Fanuc TP program (LS listing): model4_recl.ls

/PROG  model4_recl
/ATTR
COMMENT	= "19-03-19 17:59:41";
PROG_SIZE	= 0;
DEFAULT_GROUP	= 1, *, *, *, *;
/APPL
    ARC Welding Equipment: 1, *, *, *, *;
/MN
   1:  CALL HOME_ALL;
   1:  UFRAME_NUM = 1;
   1:  UTOOL_NUM = 3;
   1:  COL GUARD ADJUST 150;
   1:  PR[91] = PR[90];
   1:  PR[91,1] = PR[90,1] + 6.250;
   1:  PR[91,2] = PR[90,2] + 41.867;
   1:  PR[91,3] = PR[90,3] + 1.495;
   1:  PR[92] = PR[91];
   1:  PR[92,3] = PR[92,3] + 50;
   1:J PR[92] 10% FINE;
   1:L PR[91] R[100]mm/sec CNT100;
   1:  CALL LASER_DRAHT_START;
   1:  PR[91,1] = PR[90,1] + 5.356;
   1:  PR[91,2] = PR[90,2] + 42.761;
   1:L PR[91] R[100]mm/sec CNT100;
   1:  PR[91,1] = PR[90,1] + 3.853;
   1:  PR[91,2] = PR[90,2] + 48.367;
   1:L PR[91] R[100]mm/sec CNT100;
   1:  PR[91,1] = PR[90,1] + 5.356;
   1:  PR[91,2] = PR[90,2] + 53.973;
   1:L PR[91] R[100]mm/sec CNT100;
   1:  PR[91,1] = PR[90,1] + 6.250;
   1:  PR[91,2] = PR[90,2] + 54.867;
   1:L PR[91] R[100]mm/sec CNT100;
   1:  PR[91,1] = PR[90,1] + -1.119;
   1:L PR[91] R[100]mm/sec CNT100;
   1:  PR[91,1] = PR[90,1] + -0.226;
   1:  PR[91,2] = PR[90,2] + 53.973;
   1:L PR[91] R[100]mm/sec CNT100;
   1:  PR[91,1] = PR[90,1] + 1.277;
   1:  PR[91,2] = PR[90,2] + 48.367;
   1:L PR[91] R[100]mm/sec CNT100;
   1:  PR[91,1] = PR[90,1] + -0.226;
   1:  PR[91,2] = PR[90,2] + 42.761;
   1:L PR[91] R[100]mm/sec CNT100;
   1:  PR[91,1] = PR[90,1] + -1.119;
   1:  PR[91,2] = PR[90,2] + 41.867;
   1:L PR[91] R[100]mm/sec CNT100;
   1:  PR[91,1] = PR[90,1] + 6.250;
   1:L PR[91] R[100]mm/sec CNT100TB   .50sec,CALL END_PUD;
   1:  PR[92] = PR[91];
   1:  PR[92,3] = PR[92,3] + 50;
   1:J PR[92] 10% FINE;
   1:  PR[91,1] = PR[90,1] + 25.565;
   1:  PR[91,2] = PR[90,2] + 37.867;
   1:  PR[92] = PR[91];
   1:  PR[92,3] = PR[92,3] + 50;
   1:J PR[92] 10% FINE;
   1:L PR[91] R[100]mm/sec CNT100;
   1:  CALL LASER_DRAHT_START;
   1:  PR[91,2] = PR[90,2] + 58.867;
   1:L PR[91] R[100]mm/sec CNT100;
   1:  PR[91,1] = PR[90,1] + -20.435;
   1:L PR[91] R[100]mm/sec CNT100;
   1:  PR[91,2] = PR[90,2] + 37.867;
   1:L PR[91] R[100]mm/sec CNT100;
   1:  PR[91,1] = PR[90,1] + 25.565;
   1:L PR[91] R[100]mm/sec CNT100TB   .50sec,CALL END_PUD;
   1:  PR[92] = PR[91];
   1:  PR[92,3] = PR[92,3] + 50;
   1:J PR[92] 10% FINE;
   1:  PR[91,1] = PR[90,1] + 18.601;
   1:  PR[91,2] = PR[90,2] + 42.244;
   1:  PR[92] = PR[91];
   1:  PR[92,3] = PR[92,3] + 50;
   1:J PR[92] 10% FINE;
   1:L PR[91] R[100]mm/sec CNT100;
   1:  CALL LASER_DRAHT_START;
   1:  PR[91,1] = PR[90,1] + 15.065;
   1:  PR[91,2] = PR[90,2] + 41.296;
   1:L PR[91] R[100]mm/sec CNT100;
   1:  PR[91,1] = PR[90,1] + 11.530;
   1:  PR[91,2] = PR[90,2] + 42.244;
   1:L PR[91] R[100]mm/sec CNT100;
   1:  PR[91,1] = PR[90,1] + 8.942;
   1:  PR[91,2] = PR[90,2] + 44.831;
   1:L PR[91] R[100]mm/sec CNT100;
   1:  PR[91,1] = PR[90,1] + 7.995;
   1:  PR[91,2] = PR[90,2] + 48.367;
   1:L PR[91] R[100]mm/sec CNT100;
   1:  PR[91,1] = PR[90,1] + 8.942;
   1:  PR[91,2] = PR[90,2] + 51.903;
   1:L PR[91] R[100]mm/sec CNT100;
   1:  PR[91,1] = PR[90,1] + 11.530;
   1:  PR[91,2] = PR[90,2] + 54.490;
   1:L PR[91] R[100]mm/sec CNT100;
   1:  PR[91,1] = PR[90,1] + 15.065;
   1:  PR[91,2] = PR[90,2] + 55.438;
   1:L PR[91] R[100]mm/sec CNT100;
   1:  PR[91,1] = PR[90,1] + 18.601;
   1:  PR[91,2] = PR[90,2] + 54.490;
   1:L PR[91] R[100]mm/sec CNT100;
   1:  PR[91,1] = PR[90,1] + 21.188;
   1:  PR[91,2] = PR[90,2] + 51.903;
   1:L PR[91] R[100]mm/sec CNT100;
   1:  PR[91,1] = PR[90,1] + 22.136;
   1:  PR[91,2] = PR[90,2] + 48.367;
   1:L PR[91] R[100]mm/sec CNT100;
   1:  PR[91,1] = PR[90,1] + 21.188;
   1:  PR[91,2] = PR[90,2] + 44.831;
   1:L PR[91] R[100]mm/sec CNT100;
   1:  PR[91,1] = PR[90,1] + 18.601;
   1:  PR[91,2] = PR[90,2] + 42.244;
   1:L PR[91] R[100]mm/sec CNT100TB   .50sec,CALL END_PUD;
   1:  PR[92] = PR[91];
   1:  PR[92,3] = PR[92,3] + 50;
   1:J PR[92] 10% FINE;
   1:  PR[91,1] = PR[90,1] + -3.812;
   1:  PR[91,2] = PR[90,2] + 44.831;
   1:  PR[92] = PR[91];
   1:  PR[92,3] = PR[92,3] + 50;
   1:J PR[92] 10% FINE;
   1:L PR[91] R[100]mm/sec CNT100;
   1:  CALL LASER_DRAHT_START;
   1:  PR[91,1] = PR[90,1] + -6.399;
   1:  PR[91,2] = PR[90,2] + 42.244;
   1:L PR[91] R[100]mm/sec CNT100;
   1:  PR[91,1] = PR[90,1] + -9.935;
   1:  PR[91,2] = PR[90,2] + 41.296;
   1:L PR[91] R[100]mm/sec CNT100;
   1:  PR[91,1] = PR[90,1] + -13.470;
   1:  PR[91,2] = PR[90,2] + 42.244;
   1:L PR[91] R[100]mm/sec CNT100;
   1:  PR[91,1] = PR[90,1] + -16.058;
   1:  PR[91,2] = PR[90,2] + 44.831;
   1:L PR[91] R[100]mm/sec CNT100;
   1:  PR[91,1] = PR[90,1] + -17.005;
   1:  PR[91,2] = PR[90,2] + 48.367;
   1:L PR[91] R[100]mm/sec CNT100;
   1:  PR[91,1] = PR[90,1] + -16.058;
   1:  PR[91,2] = PR[90,2] + 51.903;
   1:L PR[91] R[100]mm/sec CNT100;
   1:  PR[91,1] = PR[90,1] + -13.470;
   1:  PR[91,2] = PR[90,2] + 54.490;
   1:L PR[91] R[100]mm/sec CNT100;
   1:  PR[91,1] = PR[90,1] + -9.935;
   1:  PR[91,2] = PR[90,2] + 55.438;
   1:L PR[91] R[100]mm/sec CNT100;
   1:  PR[91,1] = PR[90,1] + -6.399;
   1:  PR[91,2] = PR[90,2] + 54.490;
   1:L PR[91] R[100]mm/sec CNT100;
   1:  PR[91,1] = PR[90,1] + -3.812;
   1:  PR[91,2] = PR[90,2] + 51.903;
   1:L PR[91] R[100]mm/sec CNT100;
   1:  PR[91,1] = PR[90,1] + -2.864;
   1:  PR[91,2] = PR[90,2] + 48.367;
   1:L PR[91] R[100]mm/sec CNT100;
   1:  PR[91,1] = PR[90,1] + -3.812;
   1:  PR[91,2] = PR[90,2] + 44.831;
   1:L PR[91] R[100]mm/sec CNT100TB   .50sec,CALL END_PUD;
   1:  PR[92] = PR[91];
   1:  PR[92,3] = PR[92,3] + 50;
   1:J PR[92] 10% FINE;
   1:  PR[91] = PR[90];
   1:  PR[91,1] = PR[90,1] + 6.250;
   1:  PR[91,2] = PR[90,2] + 54.867;
   1:  PR[91,3] = PR[90,3] + 2.795;
   1:  PR[92] = PR[91];
   1:  PR[92,3] = PR[92,3] + 50;
   1:J PR[92] 10% FINE;
   1:L PR[91] R[100]mm/sec CNT100;
   1:  CALL LASER_DRAHT_START;
   1:  PR[91,1] = PR[90,1] + -1.119;
   1:L PR[91] R[100]mm/sec CNT100;
   1:  PR[91,1] = PR[90,1] + -0.226;
   1:  PR[91,2] = PR[90,2] + 53.973;
   1:L PR[91] R[100]mm/sec CNT100;
   1:  PR[91,1] = PR[90,1] + 1.277;
   1:  PR[91,2] = PR[90,2] + 48.367;
   1:L PR[91] R[100]mm/sec CNT100;
   1:  PR[91,1] = PR[90,1] + -0.226;
   1:  PR[91,2] = PR[90,2] + 42.761;
   1:L PR[91] R[100]mm/sec CNT100;
   1:  PR[91,1] = PR[90,1] + -1.119;
   1:  PR[91,2] = PR[90,2] + 41.867;
   1:L PR[91] R[100]mm/sec CNT100;
   1:  PR[91,1] = PR[90,1] + 6.250;
   1:L PR[91] R[100]mm/sec CNT100;
   1:  PR[91,1] = PR[90,1] + 5.356;
   1:  PR[91,2] = PR[90,2] + 42.761;
   1:L PR[91] R[100]mm/sec CNT100;
   1:  PR[91,1] = PR[90,1] + 3.853;
   1:  PR[91,2] = PR[90,2] + 48.367;
   1:L PR[91] R[100]mm/sec CNT100;
   1:  PR[91,1] = PR[90,1] + 5.356;
   1:  PR[91,2] = PR[90,2] + 53.973;
   1:L PR[91] R[100]mm/sec CNT100;
   1:  PR[91,1] = PR[90,1] + 6.250;
   1:  PR[91,2] = PR[90,2] + 54.867;
   1:L PR[91] R[100]mm/sec CNT100TB   .50sec,CALL END_PUD;
   1:  PR[92] = PR[91];
   1:  PR[92,3] = PR[92,3] + 50;
   1:J PR[92] 10% FINE;
   1:  PR[91,1] = PR[90,1] + 25.565;
   1:  PR[91,2] = PR[90,2] + 58.867;
   1:  PR[92] = PR[91];
   1:  PR[92,3] = PR[92,3] + 50;
   1:J PR[92] 10% FINE;
   1:L PR[91] R[100]mm/sec CNT100;
   1:  CALL LASER_DRAHT_START;
   1:  PR[91,1] = PR[90,1] + -20.435;
   1:L PR[91] R[100]mm/sec CNT100;
   1:  PR[91,2] = PR[90,2] + 37.867;
   1:L PR[91] R[100]mm/sec CNT100;
   1:  PR[91,1] = PR[90,1] + 25.565;
   1:L PR[91] R[100]mm/sec CNT100;
   1:  PR[91,2] = PR[90,2] + 58.867;
   1:L PR[91] R[100]mm/sec CNT100TB   .50sec,CALL END_PUD;
   1:  PR[92] = PR[91];
   1:  PR[92,3] = PR[92,3] + 50;
   1:J PR[92] 10% FINE;
   1:  PR[91,1] = PR[90,1] + 18.601;
   1:  PR[91,2] = PR[90,2] + 54.490;
   1:  PR[92] = PR[91];
   1:  PR[92,3] = PR[92,3] + 50;
   1:J PR[92] 10% FINE;
   1:L PR[91] R[100]mm/sec CNT100;
   1:  CALL LASER_DRAHT_START;
   1:  PR[91,1] = PR[90,1] + 21.188;
   1:  PR[91,2] = PR[90,2] + 51.903;
   1:L PR[91] R[100]mm/sec CNT100;
   1:  PR[91,1] = PR[90,1] + 22.136;
   1:  PR[91,2] = PR[90,2] + 48.367;
   1:L PR[91] R[100]mm/sec CNT100;
   1:  PR[91,1] = PR[90,1] + 21.188;
   1:  PR[91,2] = PR[90,2] + 44.831;
   1:L PR[91] R[100]mm/sec CNT100;
   1:  PR[91,1] = PR[90,1] + 18.601;
   1:  PR[91,2] = PR[90,2] + 42.244;
   1:L PR[91] R[100]mm/sec CNT100;
   1:  PR[91,1] = PR[90,1] + 15.065;
   1:  PR[91,2] = PR[90,2] + 41.296;
   1:L PR[91] R[100]mm/sec CNT100;
   1:  PR[91,1] = PR[90,1] + 11.530;
   1:  PR[91,2] = PR[90,2] + 42.244;
   1:L PR[91] R[100]mm/sec CNT100;
   1:  PR[91,1] = PR[90,1] + 8.942;
   1:  PR[91,2] = PR[90,2] + 44.831;
   1:L PR[91] R[100]mm/sec CNT100;
   1:  PR[91,1] = PR[90,1] + 7.995;
   1:  PR[91,2] = PR[90,2] + 48.367;
   1:L PR[91] R[100]mm/sec CNT100;
   1:  PR[91,1] = PR[90,1] + 8.942;
   1:  PR[91,2] = PR[90,2] + 51.903;
   1:L PR[91] R[100]mm/sec CNT100;
   1:  PR[91,1] = PR[90,1] + 11.530;
   1:  PR[91,2] = PR[90,2] + 54.490;
   1:L PR[91] R[100]mm/sec CNT100;
   1:  PR[91,1] = PR[90,1] + 15.065;
   1:  PR[91,2] = PR[90,2] + 55.438;
   1:L PR[91] R[100]mm/sec CNT100;
   1:  PR[91,1] = PR[90,1] + 18.601;
   1:  PR[91,2] = PR[90,2] + 54.490;
   1:L PR[91] R[100]mm/sec CNT100TB   .50sec,CALL END_PUD;
   1:  PR[92] = PR[91];
   1:  PR[92,3] = PR[92,3] + 50;
   1:J PR[92] 10% FINE;
   1:  PR[91,1] = PR[90,1] + -3.812;
   1:  PR[91,2] = PR[90,2] + 51.903;
   1:  PR[92] = PR[91];
   1:  PR[92,3] = PR[92,3] + 50;
   1:J PR[92] 10% FINE;
   1:L PR[91] R[100]mm/sec CNT100;
   1:  CALL LASER_DRAHT_START;
   1:  PR[91,1] = PR[90,1] + -2.864;
   1:  PR[91,2] = PR[90,2] + 48.367;
   1:L PR[91] R[100]mm/sec CNT100;
   1:  PR[91,1] = PR[90,1] + -3.812;
   1:  PR[91,2] = PR[90,2] + 44.831;
   1:L PR[91] R[100]mm/sec CNT100;
   1:  PR[91,1] = PR[90,1] + -6.399;
   1:  PR[91,2] = PR[90,2] + 42.244;
   1:L PR[91] R[100]mm/sec CNT100;
   1:  PR[91,1] = PR[90,1] + -9.935;
   1:  PR[91,2] = PR[90,2] + 41.296;
   1:L PR[91] R[100]mm/sec CNT100;
   1:  PR[91,1] = PR[90,1] + -13.470;
   1:  PR[91,2] = PR[90,2] + 42.244;
   1:L PR[91] R[100]mm/sec CNT100;
   1:  PR[91,1] = PR[90,1] + -16.058;
   1:  PR[91,2] = PR[90,2] + 44.831;
   1:L PR[91] R[100]mm/sec CNT100;
   1:  PR[91,1] = PR[90,1] + -17.005;
   1:  PR[91,2] = PR[90,2] + 48.367;
   1:L PR[91] R[100]mm/sec CNT100;
   1:  PR[91,1] = PR[90,1] + -16.058;
   1:  PR[91,2] = PR[90,2] + 51.903;
   1:L PR[91] R[100]mm/sec CNT100;
   1:  PR[91,1] = PR[90,1] + -13.470;
   1:  PR[91,2] = PR[90,2] + 54.490;
   1:L PR[91] R[100]mm/sec CNT100;
   1:  PR[91,1] = PR[90,1] + -9.935;
   1:  PR[91,2] = PR[90,2] + 55.438;
   1:L PR[91] R[100]mm/sec CNT100;
   1:  PR[91,1] = PR[90,1] + -6.399;
   1:  PR[91,2] = PR[90,2] + 54.490;
   1:L PR[91] R[100]mm/sec CNT100;
   1:  PR[91,1] = PR[90,1] + -3.812;
   1:  PR[91,2] = PR[90,2] + 51.903;
   1:L PR[91] R[100]mm/sec CNT100TB   .50sec,CALL END_PUD;
   1:  PR[92] = PR[91];
   1:  PR[92,3] = PR[92,3] + 50;
   1:J PR[92] 10% FINE;
   1:  PR[91] = PR[90];
   1:  PR[91,1] = PR[90,1] + 6.250;
   1:  PR[91,2] = PR[90,2] + 54.867;
   1:  PR[91,3] = PR[90,3] + 4.095;
   1:  PR[92] = PR[91];
   1:  PR[92,3] = PR[92,3] + 50;
   1:J PR[92] 10% FINE;
   1:L PR[91] R[100]mm/sec CNT100;
   1:  CALL LASER_DRAHT_START;
   1:  PR[91,1] = PR[90,1] + -1.119;
   1:L PR[91] R[100]mm/sec CNT100;
   1:  PR[91,1] = PR[90,1] + -0.226;
   1:  PR[91,2] = PR[90,2] + 53.973;
   1:L PR[91] R[100]mm/sec CNT100;
   1:  PR[91,1] = PR[90,1] + 1.277;
   1:  PR[91,2] = PR[90,2] + 48.367;
   1:L PR[91] R[100]mm/sec CNT100;
   1:  PR[91,1] = PR[90,1] + -0.226;
   1:  PR[91,2] = PR[90,2] + 42.761;
   1:L PR[91] R[100]mm/sec CNT100;
   1:  PR[91,1] = PR[90,1] + -1.119;
   1:  PR[91,2] = PR[90,2] + 41.867;
   1:L PR[91] R[100]mm/sec CNT100;
   1:  PR[91,1] = PR[90,1] + 6.250;
   1:L PR[91] R[100]mm/sec CNT100;
   1:  PR[91,1] = PR[90,1] + 5.356;
   1:  PR[91,2] = PR[90,2] + 42.761;
   1:L PR[91] R[100]mm/sec CNT100;
   1:  PR[91,1] = PR[90,1] + 3.853;
   1:  PR[91,2] = PR[90,2] + 48.367;
   1:L PR[91] R[100]mm/sec CNT100;
   1:  PR[91,1] = PR[90,1] + 5.356;
   1:  PR[91,2] = PR[90,2] + 53.973;
   1:L PR[91] R[100]mm/sec CNT100;
   1:  PR[91,1] = PR[90,1] + 6.250;
   1:  PR[91,2] = PR[90,2] + 54.867;
   1:L PR[91] R[100]mm/sec CNT100TB   .50sec,CALL END_PUD;
   1:  PR[92] = PR[91];
   1:  PR[92,3] = PR[92,3] + 50;
   1:J PR[92] 10% FINE;
   1:  PR[91,1] = PR[90,1] + 25.565;
   1:  PR[91,2] = PR[90,2] + 58.867;
   1:  PR[92] = PR[91];
   1:  PR[92,3] = PR[92,3] + 50;
   1:J PR[92] 10% FINE;
   1:L PR[91] R[100]mm/sec CNT100;
   1:  CALL LASER_DRAHT_START;
   1:  PR[91,1] = PR[90,1] + -20.435;
   1:L PR[91] R[100]mm/sec CNT100;
   1:  PR[91,2] = PR[90,2] + 37.867;
   1:L PR[91] R[100]mm/sec CNT100;
   1:  PR[91,1] = PR[90,1] + 25.565;
   1:L PR[91] R[100]mm/sec CNT100;
   1:  PR[91,2] = PR[90,2] + 58.867;
   1:L PR[91] R[100]mm/sec CNT100TB   .50sec,CALL END_PUD;
   1:  PR[92] = PR[91];
   1:  PR[92,3] = PR[92,3] + 50;
   1:J PR[92] 10% FINE;
   1:  PR[91,1] = PR[90,1] + 21.188;
   1:  PR[91,2] = PR[90,2] + 51.903;
   1:  PR[92] = PR[91];
   1:  PR[92,3] = PR[92,3] + 50;
   1:J PR[92] 10% FINE;
   1:L PR[91] R[100]mm/sec CNT100;
   1:  CALL LASER_DRAHT_START;
   1:  PR[91,1] = PR[90,1] + 22.136;
   1:  PR[91,2] = PR[90,2] + 48.367;
   1:L PR[91] R[100]mm/sec CNT100;
   1:  PR[91,1] = PR[90,1] + 21.188;
   1:  PR[91,2] = PR[90,2] + 44.831;
   1:L PR[91] R[100]mm/sec CNT100;
   1:  PR[91,1] = PR[90,1] + 18.601;
   1:  PR[91,2] = PR[90,2] + 42.244;
   1:L PR[91] R[100]mm/sec CNT100;
   1:  PR[91,1] = PR[90,1] + 15.065;
   1:  PR[91,2] = PR[90,2] + 41.296;
   1:L PR[91] R[100]mm/sec CNT100;
   1:  PR[91,1] = PR[90,1] + 11.530;
   1:  PR[91,2] = PR[90,2] + 42.244;
   1:L PR[91] R[100]mm/sec CNT100;
   1:  PR[91,1] = PR[90,1] + 8.942;
   1:  PR[91,2] = PR[90,2] + 44.831;
   1:L PR[91] R[100]mm/sec CNT100;
   1:  PR[91,1] = PR[90,1] + 7.995;
   1:  PR[91,2] = PR[90,2] + 48.367;
   1:L PR[91] R[100]mm/sec CNT100;
   1:  PR[91,1] = PR[90,1] + 8.942;
   1:  PR[91,2] = PR[90,2] + 51.903;
   1:L PR[91] R[100]mm/sec CNT100;
   1:  PR[91,1] = PR[90,1] + 11.530;
   1:  PR[91,2] = PR[90,2] + 54.490;
   1:L PR[91] R[100]mm/sec CNT100;
   1:  PR[91,1] = PR[90,1] + 15.065;
   1:  PR[91,2] = PR[90,2] + 55.438;
   1:L PR[91] R[100]mm/sec CNT100;
   1:  PR[91,1] = PR[90,1] + 18.601;
   1:  PR[91,2] = PR[90,2] + 54.490;
   1:L PR[91] R[100]mm/sec CNT100;
   1:  PR[91,1] = PR[90,1] + 21.188;
   1:  PR[91,2] = PR[90,2] + 51.903;
   1:L PR[91] R[100]mm/sec CNT100TB   .50sec,CALL END_PUD;
   1:  PR[92] = PR[91];
   1:  PR[92,3] = PR[92,3] + 50;
   1:J PR[92] 10% FINE;
   1:  PR[91,1] = PR[90,1] + -3.812;
   1:  PR[92] = PR[91];
   1:  PR[92,3] = PR[92,3] + 50;
   1:J PR[92] 10% FINE;
   1:L PR[91] R[100]mm/sec CNT100;
   1:  CALL LASER_DRAHT_START;
   1:  PR[91,1] = PR[90,1] + -2.864;
   1:  PR[91,2] = PR[90,2] + 48.367;
   1:L PR[91] R[100]mm/sec CNT100;
   1:  PR[91,1] = PR[90,1] + -3.812;
   1:  PR[91,2] = PR[90,2] + 44.831;
   1:L PR[91] R[100]mm/sec CNT100;
   1:  PR[91,1] = PR[90,1] + -6.399;
   1:  PR[91,2] = PR[90,2] + 42.244;
   1:L PR[91] R[100]mm/sec CNT100;
   1:  PR[91,1] = PR[90,1] + -9.935;
   1:  PR[91,2] = PR[90,2] + 41.296;
   1:L PR[91] R[100]mm/sec CNT100;
   1:  PR[91,1] = PR[90,1] + -13.470;
   1:  PR[91,2] = PR[90,2] + 42.244;
   1:L PR[91] R[100]mm/sec CNT100;
   1:  PR[91,1] = PR[90,1] + -16.058;
   1:  PR[91,2] = PR[90,2] + 44.831;
   1:L PR[91] R[100]mm/sec CNT100;
   1:  PR[91,1] = PR[90,1] + -17.005;
   1:  PR[91,2] = PR[90,2] + 48.367;
   1:L PR[91] R[100]mm/sec CNT100;
   1:  PR[91,1] = PR[90,1] + -16.058;
   1:  PR[91,2] = PR[90,2] + 51.903;
   1:L PR[91] R[100]mm/sec CNT100;
   1:  PR[91,1] = PR[90,1] + -13.470;
   1:  PR[91,2] = PR[90,2] + 54.490;
   1:L PR[91] R[100]mm/sec CNT100;
   1:  PR[91,1] = PR[90,1] + -9.935;
   1:  PR[91,2] = PR[90,2] + 55.438;
   1:L PR[91] R[100]mm/sec CNT100;
   1:  PR[91,1] = PR[90,1] + -6.399;
   1:  PR[91,2] = PR[90,2] + 54.490;
   1:L PR[91] R[100]mm/sec CNT100;
   1:  PR[91,1] = PR[90,1] + -3.812;
   1:  PR[91,2] = PR[90,2] + 51.903;
   1:L PR[91] R[100]mm/sec CNT100TB   .50sec,CALL END_PUD;
   1:  PR[92] = PR[91];
   1:  PR[92,3] = PR[92,3] + 50;
   1:J PR[92] 10% FINE;
   1:  PR[91] = PR[90];
   1:  PR[91,1] = PR[90,1] + -1.119;
   1:  PR[91,2] = PR[90,2] + 41.867;
   1:  PR[91,3] = PR[90,3] + 5.395;
   1:  PR[92] = PR[91];
   1:  PR[92,3] = PR[92,3] + 50;
   1:J PR[92] 10% FINE;
   1:L PR[91] R[100]mm/sec CNT100;
   1:  CALL LASER_DRAHT_START;
   1:  PR[91,1] = PR[90,1] + 6.250;
   1:L PR[91] R[100]mm/sec CNT100;
   1:  PR[91,1] = PR[90,1] + 5.356;
   1:  PR[91,2] = PR[90,2] + 42.761;
   1:L PR[91] R[100]mm/sec CNT100;
   1:  PR[91,1] = PR[90,1] + 3.853;
   1:  PR[91,2] = PR[90,2] + 48.367;
   1:L PR[91] R[100]mm/sec CNT100;
   1:  PR[91,1] = PR[90,1] + 5.356;
   1:  PR[91,2] = PR[90,2] + 53.973;
   1:L PR[91] R[100]mm/sec CNT100;
   1:  PR[91,1] = PR[90,1] + 6.250;
   1:  PR[91,2] = PR[90,2] + 54.867;
   1:L PR[91] R[100]mm/sec CNT100;
   1:  PR[91,1] = PR[90,1] + -1.119;
   1:L PR[91] R[100]mm/sec CNT100;
   1:  PR[91,1] = PR[90,1] + -0.226;
   1:  PR[91,2] = PR[90,2] + 53.973;
   1:L PR[91] R[100]mm/sec CNT100;
   1:  PR[91,1] = PR[90,1] + 1.277;
   1:  PR[91,2] = PR[90,2] + 48.367;
   1:L PR[91] R[100]mm/sec CNT100;
   1:  PR[91,1] = PR[90,1] + -0.226;
   1:  PR[91,2] = PR[90,2] + 42.761;
   1:L PR[91] R[100]mm/sec CNT100;
   1:  PR[91,1] = PR[90,1] + -1.119;
   1:  PR[91,2] = PR[90,2] + 41.867;
   1:L PR[91] R[100]mm/sec CNT100TB   .50sec,CALL END_PUD;
   1:  PR[92] = PR[91];
   1:  PR[92,3] = PR[92,3] + 50;
   1:J PR[92] 10% FINE;
   1:  PR[91,1] = PR[90,1] + -20.435;
   1:  PR[91,2] = PR[90,2] + 37.867;
   1:  PR[92] = PR[91];
   1:  PR[92,3] = PR[92,3] + 50;
   1:J PR[92] 10% FINE;
   1:L PR[91] R[100]mm/sec CNT100;
   1:  CALL LASER_DRAHT_START;
   1:  PR[91,1] = PR[90,1] + 25.565;
   1:L PR[91] R[100]mm/sec CNT100;
   1:  PR[91,2] = PR[90,2] + 58.867;
   1:L PR[91] R[100]mm/sec CNT100;
   1:  PR[91,1] = PR[90,1] + -20.435;
   1:L PR[91] R[100]mm/sec CNT100;
   1:  PR[91,2] = PR[90,2] + 37.867;
   1:L PR[91] R[100]mm/sec CNT100TB   .50sec,CALL END_PUD;
   1:  PR[92] = PR[91];
   1:  PR[92,3] = PR[92,3] + 50;
   1:J PR[92] 10% FINE;
   1:  PR[91,1] = PR[90,1] + -16.058;
   1:  PR[91,2] = PR[90,2] + 44.831;
   1:  PR[92] = PR[91];
   1:  PR[92,3] = PR[92,3] + 50;
   1:J PR[92] 10% FINE;
   1:L PR[91] R[100]mm/sec CNT100;
   1:  CALL LASER_DRAHT_START;
   1:  PR[91,1] = PR[90,1] + -17.005;
   1:  PR[91,2] = PR[90,2] + 48.367;
   1:L PR[91] R[100]mm/sec CNT100;
   1:  PR[91,1] = PR[90,1] + -16.058;
   1:  PR[91,2] = PR[90,2] + 51.903;
   1:L PR[91] R[100]mm/sec CNT100;
   1:  PR[91,1] = PR[90,1] + -13.470;
   1:  PR[91,2] = PR[90,2] + 54.490;
   1:L PR[91] R[100]mm/sec CNT100;
   1:  PR[91,1] = PR[90,1] + -9.935;
   1:  PR[91,2] = PR[90,2] + 55.438;
   1:L PR[91] R[100]mm/sec CNT100;
   1:  PR[91,1] = PR[90,1] + -6.399;
   1:  PR[91,2] = PR[90,2] + 54.490;
   1:L PR[91] R[100]mm/sec CNT100;
   1:  PR[91,1] = PR[90,1] + -3.812;
   1:  PR[91,2] = PR[90,2] + 51.903;
   1:L PR[91] R[100]mm/sec CNT100;
   1:  PR[91,1] = PR[90,1] + -2.864;
   1:  PR[91,2] = PR[90,2] + 48.367;
   1:L PR[91] R[100]mm/sec CNT100;
   1:  PR[91,1] = PR[90,1] + -3.812;
   1:  PR[91,2] = PR[90,2] + 44.831;
   1:L PR[91] R[100]mm/sec CNT100;
   1:  PR[91,1] = PR[90,1] + -6.399;
   1:  PR[91,2] = PR[90,2] + 42.244;
   1:L PR[91] R[100]mm/sec CNT100;
   1:  PR[91,1] = PR[90,1] + -9.935;
   1:  PR[91,2] = PR[90,2] + 41.296;
   1:L PR[91] R[100]mm/sec CNT100;
   1:  PR[91,1] = PR[90,1] + -13.470;
   1:  PR[91,2] = PR[90,2] + 42.244;
   1:L PR[91] R[100]mm/sec CNT100;
   1:  PR[91,1] = PR[90,1] + -16.058;
   1:  PR[91,2] = PR[90,2] + 44.831;
   1:L PR[91] R[100]mm/sec CNT100TB   .50sec,CALL END_PUD;
   1:  PR[92] = PR[91];
   1:  PR[92,3] = PR[92,3] + 50;
   1:J PR[92] 10% FINE;
   1:  PR[91,1] = PR[90,1] + 8.942;
   1:  PR[92] = PR[91];
   1:  PR[92,3] = PR[92,3] + 50;
   1:J PR[92] 10% FINE;
   1:L PR[91] R[100]mm/sec CNT100;
   1:  CALL LASER_DRAHT_START;
   1:  PR[91,1] = PR[90,1] + 7.995;
   1:  PR[91,2] = PR[90,2] + 48.367;
   1:L PR[91] R[100]mm/sec CNT100;
   1:  PR[91,1] = PR[90,1] + 8.942;
   1:  PR[91,2] = PR[90,2] + 51.903;
   1:L PR[91] R[100]mm/sec CNT100;
   1:  PR[91,1] = PR[90,1] + 11.530;
   1:  PR[91,2] = PR[90,2] + 54.490;
   1:L PR[91] R[100]mm/sec CNT100;
   1:  PR[91,1] = PR[90,1] + 15.065;
   1:  PR[91,2] = PR[90,2] + 55.438;
   1:L PR[91] R[100]mm/sec CNT100;
   1:  PR[91,1] = PR[90,1] + 18.601;
   1:  PR[91,2] = PR[90,2] + 54.490;
   1:L PR[91] R[100]mm/sec CNT100;
   1:  PR[91,1] = PR[90,1] + 21.188;
   1:  PR[91,2] = PR[90,2] + 51.903;
   1:L PR[91] R[100]mm/sec CNT100;
   1:  PR[91,1] = PR[90,1] + 22.136;
   1:  PR[91,2] = PR[90,2] + 48.367;
   1:L PR[91] R[100]mm/sec CNT100;
   1:  PR[91,1] = PR[90,1] + 21.188;
   1:  PR[91,2] = PR[90,2] + 44.831;
   1:L PR[91] R[100]mm/sec CNT100;
   1:  PR[91,1] = PR[90,1] + 18.601;
   1:  PR[91,2] = PR[90,2] + 42.244;
   1:L PR[91] R[100]mm/sec CNT100;
   1:  PR[91,1] = PR[90,1] + 15.065;
   1:  PR[91,2] = PR[90,2] + 41.296;
   1:L PR[91] R[100]mm/sec CNT100;
   1:  PR[91,1] = PR[90,1] + 11.530;
   1:  PR[91,2] = PR[90,2] + 42.244;
   1:L PR[91] R[100]mm/sec CNT100;
   1:  PR[91,1] = PR[90,1] + 8.942;
   1:  PR[91,2] = PR[90,2] + 44.831;
   1:L PR[91] R[100]mm/sec CNT100TB   .50sec,CALL END_PUD;
   1:  PR[92] = PR[91];
   1:  PR[92,3] = PR[92,3] + 50;
   1:J PR[92] 10% FINE;
   1:  PR[91] = PR[90];
   1:  PR[91,1] = PR[90,1] + 6.250;
   1:  PR[91,2] = PR[90,2] + 54.867;
   1:  PR[91,3] = PR[90,3] + 6.695;
   1:  PR[92] = PR[91];
   1:  PR[92,3] = PR[92,3] + 50;
   1:J PR[92] 10% FINE;
   1:L PR[91] R[100]mm/sec CNT100;
   1:  CALL LASER_DRAHT_START;
   1:  PR[91,1] = PR[90,1] + -1.119;
   1:L PR[91] R[100]mm/sec CNT100;
   1:  PR[91,1] = PR[90,1] + -0.226;
   1:  PR[91,2] = PR[90,2] + 53.973;
   1:L PR[91] R[100]mm/sec CNT100;
   1:  PR[91,1] = PR[90,1] + 1.277;
   1:  PR[91,2] = PR[90,2] + 48.367;
   1:L PR[91] R[100]mm/sec CNT100;
   1:  PR[91,1] = PR[90,1] + -0.226;
   1:  PR[91,2] = PR[90,2] + 42.761;
   1:L PR[91] R[100]mm/sec CNT100;
   1:  PR[91,1] = PR[90,1] + -1.119;
   1:  PR[91,2] = PR[90,2] + 41.867;
   1:L PR[91] R[100]mm/sec CNT100;
   1:  PR[91,1] = PR[90,1] + 6.250;
   1:L PR[91] R[100]mm/sec CNT100;
   1:  PR[91,1] = PR[90,1] + 5.356;
   1:  PR[91,2] = PR[90,2] + 42.761;
   1:L PR[91] R[100]mm/sec CNT100;
   1:  PR[91,1] = PR[90,1] + 3.853;
   1:  PR[91,2] = PR[90,2] + 48.367;
   1:L PR[91] R[100]mm/sec CNT100;
   1:  PR[91,1] = PR[90,1] + 5.356;
   1:  PR[91,2] = PR[90,2] + 53.973;
   1:L PR[91] R[100]mm/sec CNT100;
   1:  PR[91,1] = PR[90,1] + 6.250;
   1:  PR[91,2] = PR[90,2] + 54.867;
   1:L PR[91] R[100]mm/sec CNT100TB   .50sec,CALL END_PUD;
   1:  PR[92] = PR[91];
   1:  PR[92,3] = PR[92,3] + 50;
   1:J PR[92] 10% FINE;
   1:  PR[91,1] = PR[90,1] + 25.565;
   1:  PR[91,2] = PR[90,2] + 58.867;
   1:  PR[92] = PR[91];
   1:  PR[92,3] = PR[92,3] + 50;
   1:J PR[92] 10% FINE;
   1:L PR[91] R[100]mm/sec CNT100;
   1:  CALL LASER_DRAHT_START;
   1:  PR[91,1] = PR[90,1] + -20.435;
   1:L PR[91] R[100]mm/sec CNT100;
   1:  PR[91,2] = PR[90,2] + 37.867;
   1:L PR[91] R[100]mm/sec CNT100;
   1:  PR[91,1] = PR[90,1] + 25.565;
   1:L PR[91] R[100]mm/sec CNT100;
   1:  PR[91,2] = PR[90,2] + 58.867;
   1:L PR[91] R[100]mm/sec CNT100TB   .50sec,CALL END_PUD;
   1:  PR[92] = PR[91];
   1:  PR[92,3] = PR[92,3] + 50;
   1:J PR[92] 10% FINE;
   1:  PR[91,1] = PR[90,1] + 21.188;
   1:  PR[91,2] = PR[90,2] + 51.903;
   1:  PR[92] = PR[91];
   1:  PR[92,3] = PR[92,3] + 50;
   1:J PR[92] 10% FINE;
   1:L PR[91] R[100]mm/sec CNT100;
   1:  CALL LASER_DRAHT_START;
   1:  PR[91,1] = PR[90,1] + 22.136;
   1:  PR[91,2] = PR[90,2] + 48.367;
   1:L PR[91] R[100]mm/sec CNT100;
   1:  PR[91,1] = PR[90,1] + 21.188;
   1:  PR[91,2] = PR[90,2] + 44.831;
   1:L PR[91] R[100]mm/sec CNT100;
   1:  PR[91,1] = PR[90,1] + 18.601;
   1:  PR[91,2] = PR[90,2] + 42.244;
   1:L PR[91] R[100]mm/sec CNT100;
   1:  PR[91,1] = PR[90,1] + 15.065;
   1:  PR[91,2] = PR[90,2] + 41.296;
   1:L PR[91] R[100]mm/sec CNT100;
   1:  PR[91,1] = PR[90,1] + 11.530;
   1:  PR[91,2] = PR[90,2] + 42.244;
   1:L PR[91] R[100]mm/sec CNT100;
   1:  PR[91,1] = PR[90,1] + 8.942;
   1:  PR[91,2] = PR[90,2] + 44.831;
   1:L PR[91] R[100]mm/sec CNT100;
   1:  PR[91,1] = PR[90,1] + 7.995;
   1:  PR[91,2] = PR[90,2] + 48.367;
   1:L PR[91] R[100]mm/sec CNT100;
   1:  PR[91,1] = PR[90,1] + 8.942;
   1:  PR[91,2] = PR[90,2] + 51.903;
   1:L PR[91] R[100]mm/sec CNT100;
   1:  PR[91,1] = PR[90,1] + 11.530;
   1:  PR[91,2] = PR[90,2] + 54.490;
   1:L PR[91] R[100]mm/sec CNT100;
   1:  PR[91,1] = PR[90,1] + 15.065;
   1:  PR[91,2] = PR[90,2] + 55.438;
   1:L PR[91] R[100]mm/sec CNT100;
   1:  PR[91,1] = PR[90,1] + 18.601;
   1:  PR[91,2] = PR[90,2] + 54.490;
   1:L PR[91] R[100]mm/sec CNT100;
   1:  PR[91,1] = PR[90,1] + 21.188;
   1:  PR[91,2] = PR[90,2] + 51.903;
   1:L PR[91] R[100]mm/sec CNT100TB   .50sec,CALL END_PUD;
   1:  PR[92] = PR[91];
   1:  PR[92,3] = PR[92,3] + 50;
   1:J PR[92] 10% FINE;
   1:  PR[91,1] = PR[90,1] + -3.812;
   1:  PR[92] = PR[91];
   1:  PR[92,3] = PR[92,3] + 50;
   1:J PR[92] 10% FINE;
   1:L PR[91] R[100]mm/sec CNT100;
   1:  CALL LASER_DRAHT_START;
   1:  PR[91,1] = PR[90,1] + -2.864;
   1:  PR[91,2] = PR[90,2] + 48.367;
   1:L PR[91] R[100]mm/sec CNT100;
   1:  PR[91,1] = PR[90,1] + -3.812;
   1:  PR[91,2] = PR[90,2] + 44.831;
   1:L PR[91] R[100]mm/sec CNT100;
   1:  PR[91,1] = PR[90,1] + -6.399;
   1:  PR[91,2] = PR[90,2] + 42.244;
   1:L PR[91] R[100]mm/sec CNT100;
   1:  PR[91,1] = PR[90,1] + -9.935;
   1:  PR[91,2] = PR[90,2] + 41.296;
   1:L PR[91] R[100]mm/sec CNT100;
   1:  PR[91,1] = PR[90,1] + -13.470;
   1:  PR[91,2] = PR[90,2] + 42.244;
   1:L PR[91] R[100]mm/sec CNT100;
   1:  PR[91,1] = PR[90,1] + -16.058;
   1:  PR[91,2] = PR[90,2] + 44.831;
   1:L PR[91] R[100]mm/sec CNT100;
   1:  PR[91,1] = PR[90,1] + -17.005;
   1:  PR[91,2] = PR[90,2] + 48.367;
   1:L PR[91] R[100]mm/sec CNT100;
   1:  PR[91,1] = PR[90,1] + -16.058;
   1:  PR[91,2] = PR[90,2] + 51.903;
   1:L PR[91] R[100]mm/sec CNT100;
   1:  PR[91,1] = PR[90,1] + -13.470;
   1:  PR[91,2] = PR[90,2] + 54.490;
   1:L PR[91] R[100]mm/sec CNT100;
   1:  PR[91,1] = PR[90,1] + -9.935;
   1:  PR[91,2] = PR[90,2] + 55.438;
   1:L PR[91] R[100]mm/sec CNT100;
   1:  PR[91,1] = PR[90,1] + -6.399;
   1:  PR[91,2] = PR[90,2] + 54.490;
   1:L PR[91] R[100]mm/sec CNT100;
   1:  PR[91,1] = PR[90,1] + -3.812;
   1:  PR[91,2] = PR[90,2] + 51.903;
   1:L PR[91] R[100]mm/sec CNT100TB   .50sec,CALL END_PUD;
   1:  PR[92] = PR[91];
   1:  PR[92,3] = PR[92,3] + 50;
   1:J PR[92] 10% FINE;
   1:  PR[91] = PR[90];
   1:  PR[91,1] = PR[90,1] + -1.119;
   1:  PR[91,2] = PR[90,2] + 54.867;
   1:  PR[91,3] = PR[90,3] + 7.995;
   1:  PR[92] = PR[91];
   1:  PR[92,3] = PR[92,3] + 50;
   1:J PR[92] 10% FINE;
   1:L PR[91] R[100]mm/sec CNT100;
   1:  CALL LASER_DRAHT_START;
   1:  PR[91,1] = PR[90,1] + -0.226;
   1:  PR[91,2] = PR[90,2] + 53.973;
   1:L PR[91] R[100]mm/sec CNT100;
   1:  PR[91,1] = PR[90,1] + 1.277;
   1:  PR[91,2] = PR[90,2] + 48.367;
   1:L PR[91] R[100]mm/sec CNT100;
   1:  PR[91,1] = PR[90,1] + -0.226;
   1:  PR[91,2] = PR[90,2] + 42.761;
   1:L PR[91] R[100]mm/sec CNT100;
   1:  PR[91,1] = PR[90,1] + -1.119;
   1:  PR[91,2] = PR[90,2] + 41.867;
   1:L PR[91] R[100]mm/sec CNT100;
   1:  PR[91,1] = PR[90,1] + 6.250;
   1:L PR[91] R[100]mm/sec CNT100;
   1:  PR[91,1] = PR[90,1] + 5.356;
   1:  PR[91,2] = PR[90,2] + 42.761;
   1:L PR[91] R[100]mm/sec CNT100;
   1:  PR[91,1] = PR[90,1] + 3.853;
   1:  PR[91,2] = PR[90,2] + 48.367;
   1:L PR[91] R[100]mm/sec CNT100;
   1:  PR[91,1] = PR[90,1] + 5.356;
   1:  PR[91,2] = PR[90,2] + 53.973;
   1:L PR[91] R[100]mm/sec CNT100;
   1:  PR[91,1] = PR[90,1] + 6.250;
   1:  PR[91,2] = PR[90,2] + 54.867;
   1:L PR[91] R[100]mm/sec CNT100;
   1:  PR[91,1] = PR[90,1] + -1.119;
   1:L PR[91] R[100]mm/sec CNT100TB   .50sec,CALL END_PUD;
   1:  PR[92] = PR[91];
   1:  PR[92,3] = PR[92,3] + 50;
   1:J PR[92] 10% FINE;
   1:  PR[91,1] = PR[90,1] + -20.435;
   1:  PR[91,2] = PR[90,2] + 58.867;
   1:  PR[92] = PR[91];
   1:  PR[92,3] = PR[92,3] + 50;
   1:J PR[92] 10% FINE;
   1:L PR[91] R[100]mm/sec CNT100;
   1:  CALL LASER_DRAHT_START;
   1:  PR[91,2] = PR[90,2] + 37.867;
   1:L PR[91] R[100]mm/sec CNT100;
   1:  PR[91,1] = PR[90,1] + 25.565;
   1:L PR[91] R[100]mm/sec CNT100;
   1:  PR[91,2] = PR[90,2] + 58.867;
   1:L PR[91] R[100]mm/sec CNT100;
   1:  PR[91,1] = PR[90,1] + -20.435;
   1:L PR[91] R[100]mm/sec CNT100TB   .50sec,CALL END_PUD;
   1:  PR[92] = PR[91];
   1:  PR[92,3] = PR[92,3] + 50;
   1:J PR[92] 10% FINE;
   1:  PR[91,1] = PR[90,1] + -13.470;
   1:  PR[91,2] = PR[90,2] + 54.490;
   1:  PR[92] = PR[91];
   1:  PR[92,3] = PR[92,3] + 50;
   1:J PR[92] 10% FINE;
   1:L PR[91] R[100]mm/sec CNT100;
   1:  CALL LASER_DRAHT_START;
   1:  PR[91,1] = PR[90,1] + -9.935;
   1:  PR[91,2] = PR[90,2] + 55.438;
   1:L PR[91] R[100]mm/sec CNT100;
   1:  PR[91,1] = PR[90,1] + -6.399;
   1:  PR[91,2] = PR[90,2] + 54.490;
   1:L PR[91] R[100]mm/sec CNT100;
   1:  PR[91,1] = PR[90,1] + -3.812;
   1:  PR[91,2] = PR[90,2] + 51.903;
   1:L PR[91] R[100]mm/sec CNT100;
   1:  PR[91,1] = PR[90,1] + -2.864;
   1:  PR[91,2] = PR[90,2] + 48.367;
   1:L PR[91] R[100]mm/sec CNT100;
   1:  PR[91,1] = PR[90,1] + -3.812;
   1:  PR[91,2] = PR[90,2] + 44.831;
   1:L PR[91] R[100]mm/sec CNT100;
   1:  PR[91,1] = PR[90,1] + -6.399;
   1:  PR[91,2] = PR[90,2] + 42.244;
   1:L PR[91] R[100]mm/sec CNT100;
   1:  PR[91,1] = PR[90,1] + -9.935;
   1:  PR[91,2] = PR[90,2] + 41.296;
   1:L PR[91] R[100]mm/sec CNT100;
   1:  PR[91,1] = PR[90,1] + -13.470;
   1:  PR[91,2] = PR[90,2] + 42.244;
   1:L PR[91] R[100]mm/sec CNT100;
   1:  PR[91,1] = PR[90,1] + -16.058;
   1:  PR[91,2] = PR[90,2] + 44.831;
   1:L PR[91] R[100]mm/sec CNT100;
   1:  PR[91,1] = PR[90,1] + -17.005;
   1:  PR[91,2] = PR[90,2] + 48.367;
   1:L PR[91] R[100]mm/sec CNT100;
   1:  PR[91,1] = PR[90,1] + -16.058;
   1:  PR[91,2] = PR[90,2] + 51.903;
   1:L PR[91] R[100]mm/sec CNT100;
   1:  PR[91,1] = PR[90,1] + -13.470;
   1:  PR[91,2] = PR[90,2] + 54.490;
   1:L PR[91] R[100]mm/sec CNT100TB   .50sec,CALL END_PUD;
   1:  PR[92] = PR[91];
   1:  PR[92,3] = PR[92,3] + 50;
   1:J PR[92] 10% FINE;
   1:  PR[91,1] = PR[90,1] + 8.942;
   1:  PR[91,2] = PR[90,2] + 51.903;
   1:  PR[92] = PR[91];
   1:  PR[92,3] = PR[92,3] + 50;
   1:J PR[92] 10% FINE;
   1:L PR[91] R[100]mm/sec CNT100;
   1:  CALL LASER_DRAHT_START;
   1:  PR[91,1] = PR[90,1] + 11.530;
   1:  PR[91,2] = PR[90,2] + 54.490;
   1:L PR[91] R[100]mm/sec CNT100;
   1:  PR[91,1] = PR[90,1] + 15.065;
   1:  PR[91,2] = PR[90,2] + 55.438;
   1:L PR[91] R[100]mm/sec CNT100;
   1:  PR[91,1] = PR[90,1] + 18.601;
   1:  PR[91,2] = PR[90,2] + 54.490;
   1:L PR[91] R[100]mm/sec CNT100;
   1:  PR[91,1] = PR[90,1] + 21.188;
   1:  PR[91,2] = PR[90,2] + 51.903;
   1:L PR[91] R[100]mm/sec CNT100;
   1:  PR[91,1] = PR[90,1] + 22.136;
   1:  PR[91,2] = PR[90,2] + 48.367;
   1:L PR[91] R[100]mm/sec CNT100;
   1:  PR[91,1] = PR[90,1] + 21.188;
   1:  PR[91,2] = PR[90,2] + 44.831;
   1:L PR[91] R[100]mm/sec CNT100;
   1:  PR[91,1] = PR[90,1] + 18.601;
   1:  PR[91,2] = PR[90,2] + 42.244;
   1:L PR[91] R[100]mm/sec CNT100;
   1:  PR[91,1] = PR[90,1] + 15.065;
   1:  PR[91,2] = PR[90,2] + 41.296;
   1:L PR[91] R[100]mm/sec CNT100;
   1:  PR[91,1] = PR[90,1] + 11.530;
   1:  PR[91,2] = PR[90,2] + 42.244;
   1:L PR[91] R[100]mm/sec CNT100;
   1:  PR[91,1] = PR[90,1] + 8.942;
   1:  PR[91,2] = PR[90,2] + 44.831;
   1:L PR[91] R[100]mm/sec CNT100;
   1:  PR[91,1] = PR[90,1] + 7.995;
   1:  PR[91,2] = PR[90,2] + 48.367;
   1:L PR[91] R[100]mm/sec CNT100;
   1:  PR[91,1] = PR[90,1] + 8.942;
   1:  PR[91,2] = PR[90,2] + 51.903;
   1:L PR[91] R[100]mm/sec CNT100TB   .50sec,CALL END_PUD;
   1:  PR[92] = PR[91];
   1:  PR[92,3] = PR[92,3] + 50;
   1:J PR[92] 10% FINE;
   1:  PR[91] = PR[90];
   1:  PR[91,1] = PR[90,1] + 6.250;
   1:  PR[91,2] = PR[90,2] + 41.867;
   1:  PR[91,3] = PR[90,3] + 9.295;
   1:  PR[92] = PR[91];
   1:  PR[92,3] = PR[92,3] + 50;
   1:J PR[92] 10% FINE;
   1:L PR[91] R[100]mm/sec CNT100;
   1:  CALL LASER_DRAHT_START;
   1:  PR[91,1] = PR[90,1] + 5.356;
   1:  PR[91,2] = PR[90,2] + 42.761;
   1:L PR[91] R[100]mm/sec CNT100;
   1:  PR[91,1] = PR[90,1] + 3.853;
   1:  PR[91,2] = PR[90,2] + 48.367;
   1:L PR[91] R[100]mm/sec CNT100;
   1:  PR[91,1] = PR[90,1] + 5.356;
   1:  PR[91,2] = PR[90,2] + 53.973;
   1:L PR[91] R[100]mm/sec CNT100;
   1:  PR[91,1] = PR[90,1] + 6.250;
   1:  PR[91,2] = PR[90,2] + 54.867;
   1:L PR[91] R[100]mm/sec CNT100;
   1:  PR[91,1] = PR[90,1] + -1.119;
   1:L PR[91] R[100]mm/sec CNT100;
   1:  PR[91,1] = PR[90,1] + -0.226;
   1:  PR[91,2] = PR[90,2] + 53.973;
   1:L PR[91] R[100]mm/sec CNT100;
   1:  PR[91,1] = PR[90,1] + 1.277;
   1:  PR[91,2] = PR[90,2] + 48.367;
   1:L PR[91] R[100]mm/sec CNT100;
   1:  PR[91,1] = PR[90,1] + -0.226;
   1:  PR[91,2] = PR[90,2] + 42.761;
   1:L PR[91] R[100]mm/sec CNT100;
   1:  PR[91,1] = PR[90,1] + -1.119;
   1:  PR[91,2] = PR[90,2] + 41.867;
   1:L PR[91] R[100]mm/sec CNT100;
   1:  PR[91,1] = PR[90,1] + 6.250;
   1:L PR[91] R[100]mm/sec CNT100TB   .50sec,CALL END_PUD;
   1:  PR[92] = PR[91];
   1:  PR[92,3] = PR[92,3] + 50;
   1:J PR[92] 10% FINE;
   1:  PR[91,1] = PR[90,1] + 25.565;
   1:  PR[91,2] = PR[90,2] + 37.867;
   1:  PR[92] = PR[91];
   1:  PR[92,3] = PR[92,3] + 50;
   1:J PR[92] 10% FINE;
   1:L PR[91] R[100]mm/sec CNT100;
   1:  CALL LASER_DRAHT_START;
   1:  PR[91,2] = PR[90,2] + 58.867;
   1:L PR[91] R[100]mm/sec CNT100;
   1:  PR[91,1] = PR[90,1] + -20.435;
   1:L PR[91] R[100]mm/sec CNT100;
   1:  PR[91,2] = PR[90,2] + 37.867;
   1:L PR[91] R[100]mm/sec CNT100;
   1:  PR[91,1] = PR[90,1] + 25.565;
   1:L PR[91] R[100]mm/sec CNT100TB   .50sec,CALL END_PUD;
   1:  PR[92] = PR[91];
   1:  PR[92,3] = PR[92,3] + 50;
   1:J PR[92] 10% FINE;
   1:  PR[91,1] = PR[90,1] + 21.188;
   1:  PR[91,2] = PR[90,2] + 44.831;
   1:  PR[92] = PR[91];
   1:  PR[92,3] = PR[92,3] + 50;
   1:J PR[92] 10% FINE;
   1:L PR[91] R[100]mm/sec CNT100;
   1:  CALL LASER_DRAHT_START;
   1:  PR[91,1] = PR[90,1] + 18.601;
   1:  PR[91,2] = PR[90,2] + 42.244;
   1:L PR[91] R[100]mm/sec CNT100;
   1:  PR[91,1] = PR[90,1] + 15.065;
   1:  PR[91,2] = PR[90,2] + 41.296;
   1:L PR[91] R[100]mm/sec CNT100;
   1:  PR[91,1] = PR[90,1] + 11.530;
   1:  PR[91,2] = PR[90,2] + 42.244;
   1:L PR[91] R[100]mm/sec CNT100;
   1:  PR[91,1] = PR[90,1] + 8.942;
   1:  PR[91,2] = PR[90,2] + 44.831;
   1:L PR[91] R[100]mm/sec CNT100;
   1:  PR[91,1] = PR[90,1] + 7.995;
   1:  PR[91,2] = PR[90,2] + 48.367;
   1:L PR[91] R[100]mm/sec CNT100;
   1:  PR[91,1] = PR[90,1] + 8.942;
   1:  PR[91,2] = PR[90,2] + 51.903;
   1:L PR[91] R[100]mm/sec CNT100;
   1:  PR[91,1] = PR[90,1] + 11.530;
   1:  PR[91,2] = PR[90,2] + 54.490;
   1:L PR[91] R[100]mm/sec CNT100;
   1:  PR[91,1] = PR[90,1] + 15.065;
   1:  PR[91,2] = PR[90,2] + 55.438;
   1:L PR[91] R[100]mm/sec CNT100;
   1:  PR[91,1] = PR[90,1] + 18.601;
   1:  PR[91,2] = PR[90,2] + 54.490;
   1:L PR[91] R[100]mm/sec CNT100;
   1:  PR[91,1] = PR[90,1] + 21.188;
   1:  PR[91,2] = PR[90,2] + 51.903;
   1:L PR[91] R[100]mm/sec CNT100;
   1:  PR[91,1] = PR[90,1] + 22.136;
   1:  PR[91,2] = PR[90,2] + 48.367;
   1:L PR[91] R[100]mm/sec CNT100;
   1:  PR[91,1] = PR[90,1] + 21.188;
   1:  PR[91,2] = PR[90,2] + 44.831;
   1:L PR[91] R[100]mm/sec CNT100TB   .50sec,CALL END_PUD;
   1:  PR[92] = PR[91];
   1:  PR[92,3] = PR[92,3] + 50;
   1:J PR[92] 10% FINE;
   1:  PR[91,1] = PR[90,1] + -3.812;
   1:  PR[92] = PR[91];
   1:  PR[92,3] = PR[92,3] + 50;
   1:J PR[92] 10% FINE;
   1:L PR[91] R[100]mm/sec CNT100;
   1:  CALL LASER_DRAHT_START;
   1:  PR[91,1] = PR[90,1] + -6.399;
   1:  PR[91,2] = PR[90,2] + 42.244;
   1:L PR[91] R[100]mm/sec CNT100;
   1:  PR[91,1] = PR[90,1] + -9.935;
   1:  PR[91,2] = PR[90,2] + 41.296;
   1:L PR[91] R[100]mm/sec CNT100;
   1:  PR[91,1] = PR[90,1] + -13.470;
   1:  PR[91,2] = PR[90,2] + 42.244;
   1:L PR[91] R[100]mm/sec CNT100;
   1:  PR[91,1] = PR[90,1] + -16.058;
   1:  PR[91,2] = PR[90,2] + 44.831;
   1:L PR[91] R[100]mm/sec CNT100;
   1:  PR[91,1] = PR[90,1] + -17.005;
   1:  PR[91,2] = PR[90,2] + 48.367;
   1:L PR[91] R[100]mm/sec CNT100;
   1:  PR[91,1] = PR[90,1] + -16.058;
   1:  PR[91,2] = PR[90,2] + 51.903;
   1:L PR[91] R[100]mm/sec CNT100;
   1:  PR[91,1] = PR[90,1] + -13.470;
   1:  PR[91,2] = PR[90,2] + 54.490;
   1:L PR[91] R[100]mm/sec CNT100;
   1:  PR[91,1] = PR[90,1] + -9.935;
   1:  PR[91,2] = PR[90,2] + 55.438;
   1:L PR[91] R[100]mm/sec CNT100;
   1:  PR[91,1] = PR[90,1] + -6.399;
   1:  PR[91,2] = PR[90,2] + 54.490;
   1:L PR[91] R[100]mm/sec CNT100;
   1:  PR[91,1] = PR[90,1] + -3.812;
   1:  PR[91,2] = PR[90,2] + 51.903;
   1:L PR[91] R[100]mm/sec CNT100;
   1:  PR[91,1] = PR[90,1] + -2.864;
   1:  PR[91,2] = PR[90,2] + 48.367;
   1:L PR[91] R[100]mm/sec CNT100;
   1:  PR[91,1] = PR[90,1] + -3.812;
   1:  PR[91,2] = PR[90,2] + 44.831;
   1:L PR[91] R[100]mm/sec CNT100TB   .50sec,CALL END_PUD;
   1:  PR[92] = PR[91];
   1:  PR[92,3] = PR[92,3] + 50;
   1:J PR[92] 10% FINE;
   1:  PR[91] = PR[90];
   1:  PR[91,1] = PR[90,1] + 6.250;
   1:  PR[91,2] = PR[90,2] + 41.867;
   1:  PR[91,3] = PR[90,3] + 10.595;
   1:  PR[92] = PR[91];
   1:  PR[92,3] = PR[92,3] + 50;
   1:J PR[92] 10% FINE;
   1:L PR[91] R[100]mm/sec CNT100;
   1:  CALL LASER_DRAHT_START;
   1:  PR[91,1] = PR[90,1] + 5.356;
   1:  PR[91,2] = PR[90,2] + 42.761;
   1:L PR[91] R[100]mm/sec CNT100;
   1:  PR[91,1] = PR[90,1] + 3.853;
   1:  PR[91,2] = PR[90,2] + 48.367;
   1:L PR[91] R[100]mm/sec CNT100;
   1:  PR[91,1] = PR[90,1] + 5.356;
   1:  PR[91,2] = PR[90,2] + 53.973;
   1:L PR[91] R[100]mm/sec CNT100;
   1:  PR[91,1] = PR[90,1] + 6.250;
   1:  PR[91,2] = PR[90,2] + 54.867;
   1:L PR[91] R[100]mm/sec CNT100;
   1:  PR[91,1] = PR[90,1] + -1.119;
   1:L PR[91] R[100]mm/sec CNT100;
   1:  PR[91,1] = PR[90,1] + -0.226;
   1:  PR[91,2] = PR[90,2] + 53.973;
   1:L PR[91] R[100]mm/sec CNT100;
   1:  PR[91,1] = PR[90,1] + 1.277;
   1:  PR[91,2] = PR[90,2] + 48.367;
   1:L PR[91] R[100]mm/sec CNT100;
   1:  PR[91,1] = PR[90,1] + -0.226;
   1:  PR[91,2] = PR[90,2] + 42.761;
   1:L PR[91] R[100]mm/sec CNT100;
   1:  PR[91,1] = PR[90,1] + -1.119;
   1:  PR[91,2] = PR[90,2] + 41.867;
   1:L PR[91] R[100]mm/sec CNT100;
   1:  PR[91,1] = PR[90,1] + 6.250;
   1:L PR[91] R[100]mm/sec CNT100TB   .50sec,CALL END_PUD;
   1:  PR[92] = PR[91];
   1:  PR[92,3] = PR[92,3] + 50;
   1:J PR[92] 10% FINE;
   1:  PR[91,1] = PR[90,1] + 25.565;
   1:  PR[91,2] = PR[90,2] + 37.867;
   1:  PR[92] = PR[91];
   1:  PR[92,3] = PR[92,3] + 50;
   1:J PR[92] 10% FINE;
   1:L PR[91] R[100]mm/sec CNT100;
   1:  CALL LASER_DRAHT_START;
   1:  PR[91,2] = PR[90,2] + 58.867;
   1:L PR[91] R[100]mm/sec CNT100;
   1:  PR[91,1] = PR[90,1] + -20.435;
   1:L PR[91] R[100]mm/sec CNT100;
   1:  PR[91,2] = PR[90,2] + 37.867;
   1:L PR[91] R[100]mm/sec CNT100;
   1:  PR[91,1] = PR[90,1] + 25.565;
   1:L PR[91] R[100]mm/sec CNT100TB   .50sec,CALL END_PUD;
   1:  PR[92] = PR[91];
   1:  PR[92,3] = PR[92,3] + 50;
   1:J PR[92] 10% FINE;
   1:  PR[91,1] = PR[90,1] + 21.188;
   1:  PR[91,2] = PR[90,2] + 44.832;
   1:  PR[92] = PR[91];
   1:  PR[92,3] = PR[92,3] + 50;
   1:J PR[92] 10% FINE;
   1:L PR[91] R[100]mm/sec CNT100;
   1:  CALL LASER_DRAHT_START;
   1:  PR[91,1] = PR[90,1] + 18.601;
   1:  PR[91,2] = PR[90,2] + 42.244;
   1:L PR[91] R[100]mm/sec CNT100;
   1:  PR[91,1] = PR[90,1] + 15.065;
   1:  PR[91,2] = PR[90,2] + 41.296;
   1:L PR[91] R[100]mm/sec CNT100;
   1:  PR[91,1] = PR[90,1] + 11.530;
   1:  PR[91,2] = PR[90,2] + 42.244;
   1:L PR[91] R[100]mm/sec CNT100;
   1:  PR[91,1] = PR[90,1] + 8.942;
   1:  PR[91,2] = PR[90,2] + 44.831;
   1:L PR[91] R[100]mm/sec CNT100;
   1:  PR[91,1] = PR[90,1] + 7.995;
   1:  PR[91,2] = PR[90,2] + 48.367;
   1:L PR[91] R[100]mm/sec CNT100;
   1:  PR[91,1] = PR[90,1] + 8.942;
   1:  PR[91,2] = PR[90,2] + 51.903;
   1:L PR[91] R[100]mm/sec CNT100;
   1:  PR[91,1] = PR[90,1] + 11.530;
   1:  PR[91,2] = PR[90,2] + 54.490;
   1:L PR[91] R[100]mm/sec CNT100;
   1:  PR[91,1] = PR[90,1] + 15.065;
   1:  PR[91,2] = PR[90,2] + 55.438;
   1:L PR[91] R[100]mm/sec CNT100;
   1:  PR[91,1] = PR[90,1] + 18.601;
   1:  PR[91,2] = PR[90,2] + 54.490;
   1:L PR[91] R[100]mm/sec CNT100;
   1:  PR[91,1] = PR[90,1] + 21.188;
   1:  PR[91,2] = PR[90,2] + 51.903;
   1:L PR[91] R[100]mm/sec CNT100;
   1:  PR[91,1] = PR[90,1] + 22.136;
   1:  PR[91,2] = PR[90,2] + 48.367;
   1:L PR[91] R[100]mm/sec CNT100;
   1:  PR[91,1] = PR[90,1] + 21.188;
   1:  PR[91,2] = PR[90,2] + 44.831;
   1:L PR[91] R[100]mm/sec CNT100TB   .50sec,CALL END_PUD;
   1:  PR[92] = PR[91];
   1:  PR[92,3] = PR[92,3] + 50;
   1:J PR[92] 10% FINE;
   1:  PR[91,1] = PR[90,1] + -3.812;
   1:  PR[91,2] = PR[90,2] + 44.832;
   1:  PR[92] = PR[91];
   1:  PR[92,3] = PR[92,3] + 50;
   1:J PR[92] 10% FINE;
   1:L PR[91] R[100]mm/sec CNT100;
   1:  CALL LASER_DRAHT_START;
   1:  PR[91,1] = PR[90,1] + -6.399;
   1:  PR[91,2] = PR[90,2] + 42.244;
   1:L PR[91] R[100]mm/sec CNT100;
   1:  PR[91,1] = PR[90,1] + -9.935;
   1:  PR[91,2] = PR[90,2] + 41.296;
   1:L PR[91] R[100]mm/sec CNT100;
   1:  PR[91,1] = PR[90,1] + -13.470;
   1:  PR[91,2] = PR[90,2] + 42.244;
   1:L PR[91] R[100]mm/sec CNT100;
   1:  PR[91,1] = PR[90,1] + -16.058;
   1:  PR[91,2] = PR[90,2] + 44.831;
   1:L PR[91] R[100]mm/sec CNT100;
   1:  PR[91,1] = PR[90,1] + -17.005;
   1:  PR[91,2] = PR[90,2] + 48.367;
   1:L PR[91] R[100]mm/sec CNT100;
   1:  PR[91,1] = PR[90,1] + -16.058;
   1:  PR[91,2] = PR[90,2] + 51.903;
   1:L PR[91] R[100]mm/sec CNT100;
   1:  PR[91,1] = PR[90,1] + -13.470;
   1:  PR[91,2] = PR[90,2] + 54.490;
   1:L PR[91] R[100]mm/sec CNT100;
   1:  PR[91,1] = PR[90,1] + -9.935;
   1:  PR[91,2] = PR[90,2] + 55.438;
   1:L PR[91] R[100]mm/sec CNT100;
   1:  PR[91,1] = PR[90,1] + -6.399;
   1:  PR[91,2] = PR[90,2] + 54.490;
   1:L PR[91] R[100]mm/sec CNT100;
   1:  PR[91,1] = PR[90,1] + -3.812;
   1:  PR[91,2] = PR[90,2] + 51.903;
   1:L PR[91] R[100]mm/sec CNT100;
   1:  PR[91,1] = PR[90,1] + -2.864;
   1:  PR[91,2] = PR[90,2] + 48.367;
   1:L PR[91] R[100]mm/sec CNT100;
   1:  PR[91,1] = PR[90,1] + -3.812;
   1:  PR[91,2] = PR[90,2] + 44.831;
   1:L PR[91] R[100]mm/sec CNT100TB   .50sec,CALL END_PUD;
   1:  PR[92] = PR[91];
   1:  PR[92,3] = PR[92,3] + 50;
   1:J PR[92] 10% FINE;
   1:  PR[91] = PR[90];
   1:  PR[91,1] = PR[90,1] + -1.119;
   1:  PR[91,2] = PR[90,2] + 41.867;
   1:  PR[91,3] = PR[90,3] + 11.895;
   1:  PR[92] = PR[91];
   1:  PR[92,3] = PR[92,3] + 50;
   1:J PR[92] 10% FINE;
   1:L PR[91] R[100]mm/sec CNT100;
   1:  CALL LASER_DRAHT_START;
   1:  PR[91,1] = PR[90,1] + 6.250;
   1:L PR[91] R[100]mm/sec CNT100;
   1:  PR[91,1] = PR[90,1] + 5.356;
   1:  PR[91,2] = PR[90,2] + 42.761;
   1:L PR[91] R[100]mm/sec CNT100;
   1:  PR[91,1] = PR[90,1] + 3.853;
   1:  PR[91,2] = PR[90,2] + 48.367;
   1:L PR[91] R[100]mm/sec CNT100;
   1:  PR[91,1] = PR[90,1] + 5.356;
   1:  PR[91,2] = PR[90,2] + 53.973;
   1:L PR[91] R[100]mm/sec CNT100;
   1:  PR[91,1] = PR[90,1] + 6.250;
   1:  PR[91,2] = PR[90,2] + 54.867;
   1:L PR[91] R[100]mm/sec CNT100;
   1:  PR[91,1] = PR[90,1] + -1.119;
   1:L PR[91] R[100]mm/sec CNT100;
   1:  PR[91,1] = PR[90,1] + -0.226;
   1:  PR[91,2] = PR[90,2] + 53.973;
   1:L PR[91] R[100]mm/sec CNT100;
   1:  PR[91,1] = PR[90,1] + 1.277;
   1:  PR[91,2] = PR[90,2] + 48.367;
   1:L PR[91] R[100]mm/sec CNT100;
   1:  PR[91,1] = PR[90,1] + -0.226;
   1:  PR[91,2] = PR[90,2] + 42.761;
   1:L PR[91] R[100]mm/sec CNT100;
   1:  PR[91,1] = PR[90,1] + -1.119;
   1:  PR[91,2] = PR[90,2] + 41.867;
   1:L PR[91] R[100]mm/sec CNT100TB   .50sec,CALL END_PUD;
   1:  PR[92] = PR[91];
   1:  PR[92,3] = PR[92,3] + 50;
   1:J PR[92] 10% FINE;
   1:  PR[91,1] = PR[90,1] + -20.435;
   1:  PR[91,2] = PR[90,2] + 37.867;
   1:  PR[92] = PR[91];
   1:  PR[92,3] = PR[92,3] + 50;
   1:J PR[92] 10% FINE;
   1:L PR[91] R[100]mm/sec CNT100;
   1:  CALL LASER_DRAHT_START;
   1:  PR[91,1] = PR[90,1] + 25.565;
   1:L PR[91] R[100]mm/sec CNT100;
   1:  PR[91,2] = PR[90,2] + 58.867;
   1:L PR[91] R[100]mm/sec CNT100;
   1:  PR[91,1] = PR[90,1] + -20.435;
   1:L PR[91] R[100]mm/sec CNT100;
   1:  PR[91,2] = PR[90,2] + 37.867;
   1:L PR[91] R[100]mm/sec CNT100TB   .50sec,CALL END_PUD;
   1:  PR[92] = PR[91];
   1:  PR[92,3] = PR[92,3] + 50;
   1:J PR[92] 10% FINE;
   1:  PR[91,1] = PR[90,1] + -16.058;
   1:  PR[91,2] = PR[90,2] + 44.832;
   1:  PR[92] = PR[91];
   1:  PR[92,3] = PR[92,3] + 50;
   1:J PR[92] 10% FINE;
   1:L PR[91] R[100]mm/sec CNT100;
   1:  CALL LASER_DRAHT_START;
   1:  PR[91,1] = PR[90,1] + -17.005;
   1:  PR[91,2] = PR[90,2] + 48.367;
   1:L PR[91] R[100]mm/sec CNT100;
   1:  PR[91,1] = PR[90,1] + -16.058;
   1:  PR[91,2] = PR[90,2] + 51.903;
   1:L PR[91] R[100]mm/sec CNT100;
   1:  PR[91,1] = PR[90,1] + -13.470;
   1:  PR[91,2] = PR[90,2] + 54.490;
   1:L PR[91] R[100]mm/sec CNT100;
   1:  PR[91,1] = PR[90,1] + -9.935;
   1:  PR[91,2] = PR[90,2] + 55.438;
   1:L PR[91] R[100]mm/sec CNT100;
   1:  PR[91,1] = PR[90,1] + -6.399;
   1:  PR[91,2] = PR[90,2] + 54.490;
   1:L PR[91] R[100]mm/sec CNT100;
   1:  PR[91,1] = PR[90,1] + -3.812;
   1:  PR[91,2] = PR[90,2] + 51.903;
   1:L PR[91] R[100]mm/sec CNT100;
   1:  PR[91,1] = PR[90,1] + -2.864;
   1:  PR[91,2] = PR[90,2] + 48.367;
   1:L PR[91] R[100]mm/sec CNT100;
   1:  PR[91,1] = PR[90,1] + -3.812;
   1:  PR[91,2] = PR[90,2] + 44.832;
   1:L PR[91] R[100]mm/sec CNT100;
   1:  PR[91,1] = PR[90,1] + -6.399;
   1:  PR[91,2] = PR[90,2] + 42.244;
   1:L PR[91] R[100]mm/sec CNT100;
   1:  PR[91,1] = PR[90,1] + -9.935;
   1:  PR[91,2] = PR[90,2] + 41.296;
   1:L PR[91] R[100]mm/sec CNT100;
   1:  PR[91,1] = PR[90,1] + -13.470;
   1:  PR[91,2] = PR[90,2] + 42.244;
   1:L PR[91] R[100]mm/sec CNT100;
   1:  PR[91,1] = PR[90,1] + -16.058;
   1:  PR[91,2] = PR[90,2] + 44.832;
   1:L PR[91] R[100]mm/sec CNT100TB   .50sec,CALL END_PUD;
   1:  PR[92] = PR[91];
   1:  PR[92,3] = PR[92,3] + 50;
   1:J PR[92] 10% FINE;
   1:  PR[91,1] = PR[90,1] + 8.942;
   1:  PR[92] = PR[91];
   1:  PR[92,3] = PR[92,3] + 50;
   1:J PR[92] 10% FINE;
   1:L PR[91] R[100]mm/sec CNT100;
   1:  CALL LASER_DRAHT_START;
   1:  PR[91,1] = PR[90,1] + 7.995;
   1:  PR[91,2] = PR[90,2] + 48.367;
   1:L PR[91] R[100]mm/sec CNT100;
   1:  PR[91,1] = PR[90,1] + 8.942;
   1:  PR[91,2] = PR[90,2] + 51.903;
   1:L PR[91] R[100]mm/sec CNT100;
   1:  PR[91,1] = PR[90,1] + 11.530;
   1:  PR[91,2] = PR[90,2] + 54.490;
   1:L PR[91] R[100]mm/sec CNT100;
   1:  PR[91,1] = PR[90,1] + 15.065;
   1:  PR[91,2] = PR[90,2] + 55.438;
   1:L PR[91] R[100]mm/sec CNT100;
   1:  PR[91,1] = PR[90,1] + 18.601;
   1:  PR[91,2] = PR[90,2] + 54.490;
   1:L PR[91] R[100]mm/sec CNT100;
   1:  PR[91,1] = PR[90,1] + 21.188;
   1:  PR[91,2] = PR[90,2] + 51.903;
   1:L PR[91] R[100]mm/sec CNT100;
   1:  PR[91,1] = PR[90,1] + 22.136;
   1:  PR[91,2] = PR[90,2] + 48.367;
   1:L PR[91] R[100]mm/sec CNT100;
   1:  PR[91,1] = PR[90,1] + 21.188;
   1:  PR[91,2] = PR[90,2] + 44.832;
   1:L PR[91] R[100]mm/sec CNT100;
   1:  PR[91,1] = PR[90,1] + 18.601;
   1:  PR[91,2] = PR[90,2] + 42.244;
   1:L PR[91] R[100]mm/sec CNT100;
   1:  PR[91,1] = PR[90,1] + 15.065;
   1:  PR[91,2] = PR[90,2] + 41.296;
   1:L PR[91] R[100]mm/sec CNT100;
   1:  PR[91,1] = PR[90,1] + 11.530;
   1:  PR[91,2] = PR[90,2] + 42.244;
   1:L PR[91] R[100]mm/sec CNT100;
   1:  PR[91,1] = PR[90,1] + 8.942;
   1:  PR[91,2] = PR[90,2] + 44.832;
   1:L PR[91] R[100]mm/sec CNT100TB   .50sec,CALL END_PUD;
   1:  PR[92] = PR[91];
   1:  PR[92,3] = PR[92,3] + 50;
   1:J PR[92] 10% FINE;
   1:  PR[91] = PR[90];
   1:  PR[91,1] = PR[90,1] + 6.250;
   1:  PR[91,2] = PR[90,2] + 54.867;
   1:  PR[91,3] = PR[90,3] + 13.195;
   1:  PR[92] = PR[91];
   1:  PR[92,3] = PR[92,3] + 50;
   1:J PR[92] 10% FINE;
   1:L PR[91] R[100]mm/sec CNT100;
   1:  CALL LASER_DRAHT_START;
   1:  PR[91,1] = PR[90,1] + -1.119;
   1:L PR[91] R[100]mm/sec CNT100;
   1:  PR[91,1] = PR[90,1] + -0.226;
   1:  PR[91,2] = PR[90,2] + 53.973;
   1:L PR[91] R[100]mm/sec CNT100;
   1:  PR[91,1] = PR[90,1] + 1.277;
   1:  PR[91,2] = PR[90,2] + 48.367;
   1:L PR[91] R[100]mm/sec CNT100;
   1:  PR[91,1] = PR[90,1] + -0.226;
   1:  PR[91,2] = PR[90,2] + 42.761;
   1:L PR[91] R[100]mm/sec CNT100;
   1:  PR[91,1] = PR[90,1] + -1.119;
   1:  PR[91,2] = PR[90,2] + 41.867;
   1:L PR[91] R[100]mm/sec CNT100;
   1:  PR[91,1] = PR[90,1] + 6.250;
   1:L PR[91] R[100]mm/sec CNT100;
   1:  PR[91,1] = PR[90,1] + 5.356;
   1:  PR[91,2] = PR[90,2] + 42.761;
   1:L PR[91] R[100]mm/sec CNT100;
   1:  PR[91,1] = PR[90,1] + 3.853;
   1:  PR[91,2] = PR[90,2] + 48.367;
   1:L PR[91] R[100]mm/sec CNT100;
   1:  PR[91,1] = PR[90,1] + 5.356;
   1:  PR[91,2] = PR[90,2] + 53.973;
   1:L PR[91] R[100]mm/sec CNT100;
   1:  PR[91,1] = PR[90,1] + 6.250;
   1:  PR[91,2] = PR[90,2] + 54.867;
   1:L PR[91] R[100]mm/sec CNT100TB   .50sec,CALL END_PUD;
   1:  PR[92] = PR[91];
   1:  PR[92,3] = PR[92,3] + 50;
   1:J PR[92] 10% FINE;
   1:  PR[91,1] = PR[90,1] + 25.565;
   1:  PR[91,2] = PR[90,2] + 58.867;
   1:  PR[92] = PR[91];
   1:  PR[92,3] = PR[92,3] + 50;
   1:J PR[92] 10% FINE;
   1:L PR[91] R[100]mm/sec CNT100;
   1:  CALL LASER_DRAHT_START;
   1:  PR[91,1] = PR[90,1] + -20.435;
   1:L PR[91] R[100]mm/sec CNT100;
   1:  PR[91,2] = PR[90,2] + 37.867;
   1:L PR[91] R[100]mm/sec CNT100;
   1:  PR[91,1] = PR[90,1] + 25.565;
   1:L PR[91] R[100]mm/sec CNT100;
   1:  PR[91,2] = PR[90,2] + 58.867;
   1:L PR[91] R[100]mm/sec CNT100TB   .50sec,CALL END_PUD;
   1:  PR[92] = PR[91];
   1:  PR[92,3] = PR[92,3] + 50;
   1:J PR[92] 10% FINE;
   1:  PR[91,1] = PR[90,1] + 21.188;
   1:  PR[91,2] = PR[90,2] + 51.903;
   1:  PR[92] = PR[91];
   1:  PR[92,3] = PR[92,3] + 50;
   1:J PR[92] 10% FINE;
   1:L PR[91] R[100]mm/sec CNT100;
   1:  CALL LASER_DRAHT_START;
   1:  PR[91,1] = PR[90,1] + 22.136;
   1:  PR[91,2] = PR[90,2] + 48.367;
   1:L PR[91] R[100]mm/sec CNT100;
   1:  PR[91,1] = PR[90,1] + 21.188;
   1:  PR[91,2] = PR[90,2] + 44.832;
   1:L PR[91] R[100]mm/sec CNT100;
   1:  PR[91,1] = PR[90,1] + 18.601;
   1:  PR[91,2] = PR[90,2] + 42.244;
   1:L PR[91] R[100]mm/sec CNT100;
   1:  PR[91,1] = PR[90,1] + 15.065;
   1:  PR[91,2] = PR[90,2] + 41.296;
   1:L PR[91] R[100]mm/sec CNT100;
   1:  PR[91,1] = PR[90,1] + 11.530;
   1:  PR[91,2] = PR[90,2] + 42.244;
   1:L PR[91] R[100]mm/sec CNT100;
   1:  PR[91,1] = PR[90,1] + 8.942;
   1:  PR[91,2] = PR[90,2] + 44.832;
   1:L PR[91] R[100]mm/sec CNT100;
   1:  PR[91,1] = PR[90,1] + 7.995;
   1:  PR[91,2] = PR[90,2] + 48.367;
   1:L PR[91] R[100]mm/sec CNT100;
   1:  PR[91,1] = PR[90,1] + 8.942;
   1:  PR[91,2] = PR[90,2] + 51.903;
   1:L PR[91] R[100]mm/sec CNT100;
   1:  PR[91,1] = PR[90,1] + 11.530;
   1:  PR[91,2] = PR[90,2] + 54.490;
   1:L PR[91] R[100]mm/sec CNT100;
   1:  PR[91,1] = PR[90,1] + 15.065;
   1:  PR[91,2] = PR[90,2] + 55.438;
   1:L PR[91] R[100]mm/sec CNT100;
   1:  PR[91,1] = PR[90,1] + 18.601;
   1:  PR[91,2] = PR[90,2] + 54.490;
   1:L PR[91] R[100]mm/sec CNT100;
   1:  PR[91,1] = PR[90,1] + 21.188;
   1:  PR[91,2] = PR[90,2] + 51.903;
   1:L PR[91] R[100]mm/sec CNT100TB   .50sec,CALL END_PUD;
   1:  PR[92] = PR[91];
   1:  PR[92,3] = PR[92,3] + 50;
   1:J PR[92] 10% FINE;
   1:  PR[91,1] = PR[90,1] + -3.812;
   1:  PR[92] = PR[91];
   1:  PR[92,3] = PR[92,3] + 50;
   1:J PR[92] 10% FINE;
   1:L PR[91] R[100]mm/sec CNT100;
   1:  CALL LASER_DRAHT_START;
   1:  PR[91,1] = PR[90,1] + -2.864;
   1:  PR[91,2] = PR[90,2] + 48.367;
   1:L PR[91] R[100]mm/sec CNT100;
   1:  PR[91,1] = PR[90,1] + -3.812;
   1:  PR[91,2] = PR[90,2] + 44.832;
   1:L PR[91] R[100]mm/sec CNT100;
   1:  PR[91,1] = PR[90,1] + -6.399;
   1:  PR[91,2] = PR[90,2] + 42.244;
   1:L PR[91] R[100]mm/sec CNT100;
   1:  PR[91,1] = PR[90,1] + -9.935;
   1:  PR[91,2] = PR[90,2] + 41.296;
   1:L PR[91] R[100]mm/sec CNT100;
   1:  PR[91,1] = PR[90,1] + -13.470;
   1:  PR[91,2] = PR[90,2] + 42.244;
   1:L PR[91] R[100]mm/sec CNT100;
   1:  PR[91,1] = PR[90,1] + -16.058;
   1:  PR[91,2] = PR[90,2] + 44.832;
   1:L PR[91] R[100]mm/sec CNT100;
   1:  PR[91,1] = PR[90,1] + -17.005;
   1:  PR[91,2] = PR[90,2] + 48.367;
   1:L PR[91] R[100]mm/sec CNT100;
   1:  PR[91,1] = PR[90,1] + -16.058;
   1:  PR[91,2] = PR[90,2] + 51.903;
   1:L PR[91] R[100]mm/sec CNT100;
   1:  PR[91,1] = PR[90,1] + -13.470;
   1:  PR[91,2] = PR[90,2] + 54.490;
   1:L PR[91] R[100]mm/sec CNT100;
   1:  PR[91,1] = PR[90,1] + -9.935;
   1:  PR[91,2] = PR[90,2] + 55.438;
   1:L PR[91] R[100]mm/sec CNT100;
   1:  PR[91,1] = PR[90,1] + -6.399;
   1:  PR[91,2] = PR[90,2] + 54.490;
   1:L PR[91] R[100]mm/sec CNT100;
   1:  PR[91,1] = PR[90,1] + -3.812;
   1:  PR[91,2] = PR[90,2] + 51.903;
   1:L PR[91] R[100]mm/sec CNT100TB   .50sec,CALL END_PUD;
   1:  PR[92] = PR[91];
   1:  PR[92,3] = PR[92,3] + 50;
   1:J PR[92] 10% FINE;
   1:  PR[91] = PR[90];
   1:  PR[91,1] = PR[90,1] + 6.250;
   1:  PR[91,2] = PR[90,2] + 54.867;
   1:  PR[91,3] = PR[90,3] + 14.495;
   1:  PR[92] = PR[91];
   1:  PR[92,3] = PR[92,3] + 50;
   1:J PR[92] 10% FINE;
   1:L PR[91] R[100]mm/sec CNT100;
   1:  CALL LASER_DRAHT_START;
   1:  PR[91,1] = PR[90,1] + -1.119;
   1:L PR[91] R[100]mm/sec CNT100;
   1:  PR[91,1] = PR[90,1] + -0.225;
   1:  PR[91,2] = PR[90,2] + 53.973;
   1:L PR[91] R[100]mm/sec CNT100;
   1:  PR[91,1] = PR[90,1] + 1.277;
   1:  PR[91,2] = PR[90,2] + 48.367;
   1:L PR[91] R[100]mm/sec CNT100;
   1:  PR[91,1] = PR[90,1] + -0.225;
   1:  PR[91,2] = PR[90,2] + 42.761;
   1:L PR[91] R[100]mm/sec CNT100;
   1:  PR[91,1] = PR[90,1] + -1.119;
   1:  PR[91,2] = PR[90,2] + 41.867;
   1:L PR[91] R[100]mm/sec CNT100;
   1:  PR[91,1] = PR[90,1] + 6.250;
   1:L PR[91] R[100]mm/sec CNT100;
   1:  PR[91,1] = PR[90,1] + 5.356;
   1:  PR[91,2] = PR[90,2] + 42.761;
   1:L PR[91] R[100]mm/sec CNT100;
   1:  PR[91,1] = PR[90,1] + 3.853;
   1:  PR[91,2] = PR[90,2] + 48.367;
   1:L PR[91] R[100]mm/sec CNT100;
   1:  PR[91,1] = PR[90,1] + 5.356;
   1:  PR[91,2] = PR[90,2] + 53.973;
   1:L PR[91] R[100]mm/sec CNT100;
   1:  PR[91,1] = PR[90,1] + 6.250;
   1:  PR[91,2] = PR[90,2] + 54.867;
   1:L PR[91] R[100]mm/sec CNT100TB   .50sec,CALL END_PUD;
   1:  PR[92] = PR[91];
   1:  PR[92,3] = PR[92,3] + 50;
   1:J PR[92] 10% FINE;
   1:  PR[91,1] = PR[90,1] + 25.565;
   1:  PR[91,2] = PR[90,2] + 58.867;
   1:  PR[92] = PR[91];
   1:  PR[92,3] = PR[92,3] + 50;
   1:J PR[92] 10% FINE;
   1:L PR[91] R[100]mm/sec CNT100;
   1:  CALL LASER_DRAHT_START;
   1:  PR[91,1] = PR[90,1] + -20.435;
   1:L PR[91] R[100]mm/sec CNT100;
   1:  PR[91,2] = PR[90,2] + 37.867;
   1:L PR[91] R[100]mm/sec CNT100;
   1:  PR[91,1] = PR[90,1] + 25.565;
   1:L PR[91] R[100]mm/sec CNT100;
   1:  PR[91,2] = PR[90,2] + 58.867;
   1:L PR[91] R[100]mm/sec CNT100TB   .50sec,CALL END_PUD;
   1:  PR[92] = PR[91];
   1:  PR[92,3] = PR[92,3] + 50;
   1:J PR[92] 10% FINE;
   1:  PR[91,1] = PR[90,1] + 21.188;
   1:  PR[91,2] = PR[90,2] + 51.903;
   1:  PR[92] = PR[91];
   1:  PR[92,3] = PR[92,3] + 50;
   1:J PR[92] 10% FINE;
   1:L PR[91] R[100]mm/sec CNT100;
   1:  CALL LASER_DRAHT_START;
   1:  PR[91,1] = PR[90,1] + 22.136;
   1:  PR[91,2] = PR[90,2] + 48.367;
   1:L PR[91] R[100]mm/sec CNT100;
   1:  PR[91,1] = PR[90,1] + 21.188;
   1:  PR[91,2] = PR[90,2] + 44.832;
   1:L PR[91] R[100]mm/sec CNT100;
   1:  PR[91,1] = PR[90,1] + 18.601;
   1:  PR[91,2] = PR[90,2] + 42.244;
   1:L PR[91] R[100]mm/sec CNT100;
   1:  PR[91,1] = PR[90,1] + 15.065;
   1:  PR[91,2] = PR[90,2] + 41.296;
   1:L PR[91] R[100]mm/sec CNT100;
   1:  PR[91,1] = PR[90,1] + 11.530;
   1:  PR[91,2] = PR[90,2] + 42.244;
   1:L PR[91] R[100]mm/sec CNT100;
   1:  PR[91,1] = PR[90,1] + 8.942;
   1:  PR[91,2] = PR[90,2] + 44.832;
   1:L PR[91] R[100]mm/sec CNT100;
   1:  PR[91,1] = PR[90,1] + 7.995;
   1:  PR[91,2] = PR[90,2] + 48.367;
   1:L PR[91] R[100]mm/sec CNT100;
   1:  PR[91,1] = PR[90,1] + 8.942;
   1:  PR[91,2] = PR[90,2] + 51.903;
   1:L PR[91] R[100]mm/sec CNT100;
   1:  PR[91,1] = PR[90,1] + 11.530;
   1:  PR[91,2] = PR[90,2] + 54.490;
   1:L PR[91] R[100]mm/sec CNT100;
   1:  PR[91,1] = PR[90,1] + 15.065;
   1:  PR[91,2] = PR[90,2] + 55.438;
   1:L PR[91] R[100]mm/sec CNT100;
   1:  PR[91,1] = PR[90,1] + 18.601;
   1:  PR[91,2] = PR[90,2] + 54.490;
   1:L PR[91] R[100]mm/sec CNT100;
   1:  PR[91,1] = PR[90,1] + 21.188;
   1:  PR[91,2] = PR[90,2] + 51.903;
   1:L PR[91] R[100]mm/sec CNT100TB   .50sec,CALL END_PUD;
   1:  PR[92] = PR[91];
   1:  PR[92,3] = PR[92,3] + 50;
   1:J PR[92] 10% FINE;
   1:  PR[91,1] = PR[90,1] + -3.812;
   1:  PR[92] = PR[91];
   1:  PR[92,3] = PR[92,3] + 50;
   1:J PR[92] 10% FINE;
   1:L PR[91] R[100]mm/sec CNT100;
   1:  CALL LASER_DRAHT_START;
   1:  PR[91,1] = PR[90,1] + -2.864;
   1:  PR[91,2] = PR[90,2] + 48.367;
   1:L PR[91] R[100]mm/sec CNT100;
   1:  PR[91,1] = PR[90,1] + -3.812;
   1:  PR[91,2] = PR[90,2] + 44.832;
   1:L PR[91] R[100]mm/sec CNT100;
   1:  PR[91,1] = PR[90,1] + -6.399;
   1:  PR[91,2] = PR[90,2] + 42.244;
   1:L PR[91] R[100]mm/sec CNT100;
   1:  PR[91,1] = PR[90,1] + -9.935;
   1:  PR[91,2] = PR[90,2] + 41.296;
   1:L PR[91] R[100]mm/sec CNT100;
   1:  PR[91,1] = PR[90,1] + -13.470;
   1:  PR[91,2] = PR[90,2] + 42.244;
   1:L PR[91] R[100]mm/sec CNT100;
   1:  PR[91,1] = PR[90,1] + -16.058;
   1:  PR[91,2] = PR[90,2] + 44.832;
   1:L PR[91] R[100]mm/sec CNT100;
   1:  PR[91,1] = PR[90,1] + -17.005;
   1:  PR[91,2] = PR[90,2] + 48.367;
   1:L PR[91] R[100]mm/sec CNT100;
   1:  PR[91,1] = PR[90,1] + -16.058;
   1:  PR[91,2] = PR[90,2] + 51.903;
   1:L PR[91] R[100]mm/sec CNT100;
   1:  PR[91,1] = PR[90,1] + -13.470;
   1:  PR[91,2] = PR[90,2] + 54.490;
   1:L PR[91] R[100]mm/sec CNT100;
   1:  PR[91,1] = PR[90,1] + -9.935;
   1:  PR[91,2] = PR[90,2] + 55.438;
   1:L PR[91] R[100]mm/sec CNT100;
   1:  PR[91,1] = PR[90,1] + -6.399;
   1:  PR[91,2] = PR[90,2] + 54.490;
   1:L PR[91] R[100]mm/sec CNT100;
   1:  PR[91,1] = PR[90,1] + -3.812;
   1:  PR[91,2] = PR[90,2] + 51.903;
   1:L PR[91] R[100]mm/sec CNT100TB   .50sec,CALL END_PUD;
   1:  PR[92] = PR[91];
   1:  PR[92,3] = PR[92,3] + 50;
   1:J PR[92] 10% FINE;
   1:  PR[91] = PR[90];
   1:  PR[91,1] = PR[90,1] + -1.119;
   1:  PR[91,2] = PR[90,2] + 54.867;
   1:  PR[91,3] = PR[90,3] + 15.795;
   1:  PR[92] = PR[91];
   1:  PR[92,3] = PR[92,3] + 50;
   1:J PR[92] 10% FINE;
   1:L PR[91] R[100]mm/sec CNT100;
   1:  CALL LASER_DRAHT_START;
   1:  PR[91,1] = PR[90,1] + -0.225;
   1:  PR[91,2] = PR[90,2] + 53.973;
   1:L PR[91] R[100]mm/sec CNT100;
   1:  PR[91,1] = PR[90,1] + 1.277;
   1:  PR[91,2] = PR[90,2] + 48.367;
   1:L PR[91] R[100]mm/sec CNT100;
   1:  PR[91,1] = PR[90,1] + -0.225;
   1:  PR[91,2] = PR[90,2] + 42.761;
   1:L PR[91] R[100]mm/sec CNT100;
   1:  PR[91,1] = PR[90,1] + -1.119;
   1:  PR[91,2] = PR[90,2] + 41.867;
   1:L PR[91] R[100]mm/sec CNT100;
   1:  PR[91,1] = PR[90,1] + 6.250;
   1:L PR[91] R[100]mm/sec CNT100;
   1:  PR[91,1] = PR[90,1] + 5.356;
   1:  PR[91,2] = PR[90,2] + 42.761;
   1:L PR[91] R[100]mm/sec CNT100;
   1:  PR[91,1] = PR[90,1] + 3.853;
   1:  PR[91,2] = PR[90,2] + 48.367;
   1:L PR[91] R[100]mm/sec CNT100;
   1:  PR[91,1] = PR[90,1] + 5.356;
   1:  PR[91,2] = PR[90,2] + 53.973;
   1:L PR[91] R[100]mm/sec CNT100;
   1:  PR[91,1] = PR[90,1] + 6.250;
   1:  PR[91,2] = PR[90,2] + 54.867;
   1:L PR[91] R[100]mm/sec CNT100;
   1:  PR[91,1] = PR[90,1] + -1.119;
   1:L PR[91] R[100]mm/sec CNT100TB   .50sec,CALL END_PUD;
   1:  PR[92] = PR[91];
   1:  PR[92,3] = PR[92,3] + 50;
   1:J PR[92] 10% FINE;
   1:  PR[91,1] = PR[90,1] + -20.435;
   1:  PR[91,2] = PR[90,2] + 58.867;
   1:  PR[92] = PR[91];
   1:  PR[92,3] = PR[92,3] + 50;
   1:J PR[92] 10% FINE;
   1:L PR[91] R[100]mm/sec CNT100;
   1:  CALL LASER_DRAHT_START;
   1:  PR[91,2] = PR[90,2] + 37.867;
   1:L PR[91] R[100]mm/sec CNT100;
   1:  PR[91,1] = PR[90,1] + 25.565;
   1:L PR[91] R[100]mm/sec CNT100;
   1:  PR[91,2] = PR[90,2] + 58.867;
   1:L PR[91] R[100]mm/sec CNT100;
   1:  PR[91,1] = PR[90,1] + -20.435;
   1:L PR[91] R[100]mm/sec CNT100TB   .50sec,CALL END_PUD;
   1:  PR[92] = PR[91];
   1:  PR[92,3] = PR[92,3] + 50;
   1:J PR[92] 10% FINE;
   1:  PR[91,1] = PR[90,1] + -13.470;
   1:  PR[91,2] = PR[90,2] + 54.490;
   1:  PR[92] = PR[91];
   1:  PR[92,3] = PR[92,3] + 50;
   1:J PR[92] 10% FINE;
   1:L PR[91] R[100]mm/sec CNT100;
   1:  CALL LASER_DRAHT_START;
   1:  PR[91,1] = PR[90,1] + -9.935;
   1:  PR[91,2] = PR[90,2] + 55.438;
   1:L PR[91] R[100]mm/sec CNT100;
   1:  PR[91,1] = PR[90,1] + -6.399;
   1:  PR[91,2] = PR[90,2] + 54.490;
   1:L PR[91] R[100]mm/sec CNT100;
   1:  PR[91,1] = PR[90,1] + -3.812;
   1:  PR[91,2] = PR[90,2] + 51.903;
   1:L PR[91] R[100]mm/sec CNT100;
   1:  PR[91,1] = PR[90,1] + -2.864;
   1:  PR[91,2] = PR[90,2] + 48.367;
   1:L PR[91] R[100]mm/sec CNT100;
   1:  PR[91,1] = PR[90,1] + -3.812;
   1:  PR[91,2] = PR[90,2] + 44.832;
   1:L PR[91] R[100]mm/sec CNT100;
   1:  PR[91,1] = PR[90,1] + -6.399;
   1:  PR[91,2] = PR[90,2] + 42.244;
   1:L PR[91] R[100]mm/sec CNT100;
   1:  PR[91,1] = PR[90,1] + -9.935;
   1:  PR[91,2] = PR[90,2] + 41.296;
   1:L PR[91] R[100]mm/sec CNT100;
   1:  PR[91,1] = PR[90,1] + -13.470;
   1:  PR[91,2] = PR[90,2] + 42.244;
   1:L PR[91] R[100]mm/sec CNT100;
   1:  PR[91,1] = PR[90,1] + -16.058;
   1:  PR[91,2] = PR[90,2] + 44.832;
   1:L PR[91] R[100]mm/sec CNT100;
   1:  PR[91,1] = PR[90,1] + -17.005;
   1:  PR[91,2] = PR[90,2] + 48.367;
   1:L PR[91] R[100]mm/sec CNT100;
   1:  PR[91,1] = PR[90,1] + -16.058;
   1:  PR[91,2] = PR[90,2] + 51.903;
   1:L PR[91] R[100]mm/sec CNT100;
   1:  PR[91,1] = PR[90,1] + -13.470;
   1:  PR[91,2] = PR[90,2] + 54.490;
   1:L PR[91] R[100]mm/sec CNT100TB   .50sec,CALL END_PUD;
   1:  PR[92] = PR[91];
   1:  PR[92,3] = PR[92,3] + 50;
   1:J PR[92] 10% FINE;
   1:  PR[91,1] = PR[90,1] + 8.942;
   1:  PR[91,2] = PR[90,2] + 51.903;
   1:  PR[92] = PR[91];
   1:  PR[92,3] = PR[92,3] + 50;
   1:J PR[92] 10% FINE;
   1:L PR[91] R[100]mm/sec CNT100;
   1:  CALL LASER_DRAHT_START;
   1:  PR[91,1] = PR[90,1] + 11.530;
   1:  PR[91,2] = PR[90,2] + 54.490;
   1:L PR[91] R[100]mm/sec CNT100;
   1:  PR[91,1] = PR[90,1] + 15.065;
   1:  PR[91,2] = PR[90,2] + 55.438;
   1:L PR[91] R[100]mm/sec CNT100;
   1:  PR[91,1] = PR[90,1] + 18.601;
   1:  PR[91,2] = PR[90,2] + 54.490;
   1:L PR[91] R[100]mm/sec CNT100;
   1:  PR[91,1] = PR[90,1] + 21.188;
   1:  PR[91,2] = PR[90,2] + 51.903;
   1:L PR[91] R[100]mm/sec CNT100;
   1:  PR[91,1] = PR[90,1] + 22.136;
   1:  PR[91,2] = PR[90,2] + 48.367;
   1:L PR[91] R[100]mm/sec CNT100;
   1:  PR[91,1] = PR[90,1] + 21.188;
   1:  PR[91,2] = PR[90,2] + 44.832;
   1:L PR[91] R[100]mm/sec CNT100;
   1:  PR[91,1] = PR[90,1] + 18.601;
   1:  PR[91,2] = PR[90,2] + 42.244;
   1:L PR[91] R[100]mm/sec CNT100;
   1:  PR[91,1] = PR[90,1] + 15.065;
   1:  PR[91,2] = PR[90,2] + 41.296;
   1:L PR[91] R[100]mm/sec CNT100;
   1:  PR[91,1] = PR[90,1] + 11.530;
   1:  PR[91,2] = PR[90,2] + 42.244;
   1:L PR[91] R[100]mm/sec CNT100;
   1:  PR[91,1] = PR[90,1] + 8.942;
   1:  PR[91,2] = PR[90,2] + 44.832;
   1:L PR[91] R[100]mm/sec CNT100;
   1:  PR[91,1] = PR[90,1] + 7.995;
   1:  PR[91,2] = PR[90,2] + 48.367;
   1:L PR[91] R[100]mm/sec CNT100;
   1:  PR[91,1] = PR[90,1] + 8.942;
   1:  PR[91,2] = PR[90,2] + 51.903;
   1:L PR[91] R[100]mm/sec CNT100TB   .50sec,CALL END_PUD;
   1:  PR[92] = PR[91];
   1:  PR[92,3] = PR[92,3] + 50;
   1:J PR[92] 10% FINE;
   1:  PR[91] = PR[90];
   1:  PR[91,1] = PR[90,1] + -1.119;
   1:  PR[91,2] = PR[90,2] + 41.867;
   1:  PR[91,3] = PR[90,3] + 17.095;
   1:  PR[92] = PR[91];
   1:  PR[92,3] = PR[92,3] + 50;
   1:J PR[92] 10% FINE;
   1:L PR[91] R[100]mm/sec CNT100;
   1:  CALL LASER_DRAHT_START;
   1:  PR[91,1] = PR[90,1] + 6.250;
   1:L PR[91] R[100]mm/sec CNT100;
   1:  PR[91,1] = PR[90,1] + 5.356;
   1:  PR[91,2] = PR[90,2] + 42.761;
   1:L PR[91] R[100]mm/sec CNT100;
   1:  PR[91,1] = PR[90,1] + 3.853;
   1:  PR[91,2] = PR[90,2] + 48.367;
   1:L PR[91] R[100]mm/sec CNT100;
   1:  PR[91,1] = PR[90,1] + 5.356;
   1:  PR[91,2] = PR[90,2] + 53.973;
   1:L PR[91] R[100]mm/sec CNT100;
   1:  PR[91,1] = PR[90,1] + 6.250;
   1:  PR[91,2] = PR[90,2] + 54.867;
   1:L PR[91] R[100]mm/sec CNT100;
   1:  PR[91,1] = PR[90,1] + -1.119;
   1:L PR[91] R[100]mm/sec CNT100;
   1:  PR[91,1] = PR[90,1] + -0.225;
   1:  PR[91,2] = PR[90,2] + 53.973;
   1:L PR[91] R[100]mm/sec CNT100;
   1:  PR[91,1] = PR[90,1] + 1.277;
   1:  PR[91,2] = PR[90,2] + 48.367;
   1:L PR[91] R[100]mm/sec CNT100;
   1:  PR[91,1] = PR[90,1] + -0.225;
   1:  PR[91,2] = PR[90,2] + 42.761;
   1:L PR[91] R[100]mm/sec CNT100;
   1:  PR[91,1] = PR[90,1] + -1.119;
   1:  PR[91,2] = PR[90,2] + 41.867;
   1:L PR[91] R[100]mm/sec CNT100TB   .50sec,CALL END_PUD;
   1:  PR[92] = PR[91];
   1:  PR[92,3] = PR[92,3] + 50;
   1:J PR[92] 10% FINE;
   1:  PR[91,1] = PR[90,1] + -20.435;
   1:  PR[91,2] = PR[90,2] + 37.867;
   1:  PR[92] = PR[91];
   1:  PR[92,3] = PR[92,3] + 50;
   1:J PR[92] 10% FINE;
   1:L PR[91] R[100]mm/sec CNT100;
   1:  CALL LASER_DRAHT_START;
   1:  PR[91,1] = PR[90,1] + 25.565;
   1:L PR[91] R[100]mm/sec CNT100;
   1:  PR[91,2] = PR[90,2] + 58.867;
   1:L PR[91] R[100]mm/sec CNT100;
   1:  PR[91,1] = PR[90,1] + -20.435;
   1:L PR[91] R[100]mm/sec CNT100;
   1:  PR[91,2] = PR[90,2] + 37.867;
   1:L PR[91] R[100]mm/sec CNT100TB   .50sec,CALL END_PUD;
   1:  PR[92] = PR[91];
   1:  PR[92,3] = PR[92,3] + 50;
   1:J PR[92] 10% FINE;
   1:  PR[91,1] = PR[90,1] + -13.470;
   1:  PR[91,2] = PR[90,2] + 42.244;
   1:  PR[92] = PR[91];
   1:  PR[92,3] = PR[92,3] + 50;
   1:J PR[92] 10% FINE;
   1:L PR[91] R[100]mm/sec CNT100;
   1:  CALL LASER_DRAHT_START;
   1:  PR[91,1] = PR[90,1] + -16.058;
   1:  PR[91,2] = PR[90,2] + 44.832;
   1:L PR[91] R[100]mm/sec CNT100;
   1:  PR[91,1] = PR[90,1] + -17.005;
   1:  PR[91,2] = PR[90,2] + 48.367;
   1:L PR[91] R[100]mm/sec CNT100;
   1:  PR[91,1] = PR[90,1] + -16.058;
   1:  PR[91,2] = PR[90,2] + 51.903;
   1:L PR[91] R[100]mm/sec CNT100;
   1:  PR[91,1] = PR[90,1] + -13.470;
   1:  PR[91,2] = PR[90,2] + 54.490;
   1:L PR[91] R[100]mm/sec CNT100;
   1:  PR[91,1] = PR[90,1] + -9.935;
   1:  PR[91,2] = PR[90,2] + 55.438;
   1:L PR[91] R[100]mm/sec CNT100;
   1:  PR[91,1] = PR[90,1] + -6.399;
   1:  PR[91,2] = PR[90,2] + 54.490;
   1:L PR[91] R[100]mm/sec CNT100;
   1:  PR[91,1] = PR[90,1] + -3.812;
   1:  PR[91,2] = PR[90,2] + 51.903;
   1:L PR[91] R[100]mm/sec CNT100;
   1:  PR[91,1] = PR[90,1] + -2.864;
   1:  PR[91,2] = PR[90,2] + 48.367;
   1:L PR[91] R[100]mm/sec CNT100;
   1:  PR[91,1] = PR[90,1] + -3.812;
   1:  PR[91,2] = PR[90,2] + 44.832;
   1:L PR[91] R[100]mm/sec CNT100;
   1:  PR[91,1] = PR[90,1] + -6.399;
   1:  PR[91,2] = PR[90,2] + 42.244;
   1:L PR[91] R[100]mm/sec CNT100;
   1:  PR[91,1] = PR[90,1] + -9.935;
   1:  PR[91,2] = PR[90,2] + 41.296;
   1:L PR[91] R[100]mm/sec CNT100;
   1:  PR[91,1] = PR[90,1] + -13.470;
   1:  PR[91,2] = PR[90,2] + 42.244;
   1:L PR[91] R[100]mm/sec CNT100TB   .50sec,CALL END_PUD;
   1:  PR[92] = PR[91];
   1:  PR[92,3] = PR[92,3] + 50;
   1:J PR[92] 10% FINE;
   1:  PR[91,1] = PR[90,1] + 8.942;
   1:  PR[91,2] = PR[90,2] + 44.832;
   1:  PR[92] = PR[91];
   1:  PR[92,3] = PR[92,3] + 50;
   1:J PR[92] 10% FINE;
   1:L PR[91] R[100]mm/sec CNT100;
   1:  CALL LASER_DRAHT_START;
   1:  PR[91,1] = PR[90,1] + 7.995;
   1:  PR[91,2] = PR[90,2] + 48.367;
   1:L PR[91] R[100]mm/sec CNT100;
   1:  PR[91,1] = PR[90,1] + 8.942;
   1:  PR[91,2] = PR[90,2] + 51.903;
   1:L PR[91] R[100]mm/sec CNT100;
   1:  PR[91,1] = PR[90,1] + 11.530;
   1:  PR[91,2] = PR[90,2] + 54.490;
   1:L PR[91] R[100]mm/sec CNT100;
   1:  PR[91,1] = PR[90,1] + 15.065;
   1:  PR[91,2] = PR[90,2] + 55.438;
   1:L PR[91] R[100]mm/sec CNT100;
   1:  PR[91,1] = PR[90,1] + 18.601;
   1:  PR[91,2] = PR[90,2] + 54.490;
   1:L PR[91] R[100]mm/sec CNT100;
   1:  PR[91,1] = PR[90,1] + 21.188;
   1:  PR[91,2] = PR[90,2] + 51.903;
   1:L PR[91] R[100]mm/sec CNT100;
   1:  PR[91,1] = PR[90,1] + 22.136;
   1:  PR[91,2] = PR[90,2] + 48.367;
   1:L PR[91] R[100]mm/sec CNT100;
   1:  PR[91,1] = PR[90,1] + 21.188;
   1:  PR[91,2] = PR[90,2] + 44.832;
   1:L PR[91] R[100]mm/sec CNT100;
   1:  PR[91,1] = PR[90,1] + 18.601;
   1:  PR[91,2] = PR[90,2] + 42.244;
   1:L PR[91] R[100]mm/sec CNT100;
   1:  PR[91,1] = PR[90,1] + 15.065;
   1:  PR[91,2] = PR[90,2] + 41.296;
   1:L PR[91] R[100]mm/sec CNT100;
   1:  PR[91,1] = PR[90,1] + 11.530;
   1:  PR[91,2] = PR[90,2] + 42.244;
   1:L PR[91] R[100]mm/sec CNT100;
   1:  PR[91,1] = PR[90,1] + 8.942;
   1:  PR[91,2] = PR[90,2] + 44.832;
   1:L PR[91] R[100]mm/sec CNT100TB   .50sec,CALL END_PUD;
   1:  PR[92] = PR[91];
   1:  PR[92,3] = PR[92,3] + 50;
   1:J PR[92] 10% FINE;
   1:  PR[91] = PR[90];
   1:  PR[91,1] = PR[90,1] + 6.250;
   1:  PR[91,2] = PR[90,2] + 54.867;
   1:  PR[91,3] = PR[90,3] + 18.395;
   1:  PR[92] = PR[91];
   1:  PR[92,3] = PR[92,3] + 50;
   1:J PR[92] 10% FINE;
   1:L PR[91] R[100]mm/sec CNT100;
   1:  CALL LASER_DRAHT_START;
   1:  PR[91,1] = PR[90,1] + -1.119;
   1:L PR[91] R[100]mm/sec CNT100;
   1:  PR[91,1] = PR[90,1] + -0.225;
   1:  PR[91,2] = PR[90,2] + 53.973;
   1:L PR[91] R[100]mm/sec CNT100;
   1:  PR[91,1] = PR[90,1] + 1.277;
   1:  PR[91,2] = PR[90,2] + 48.367;
   1:L PR[91] R[100]mm/sec CNT100;
   1:  PR[91,1] = PR[90,1] + -0.225;
   1:  PR[91,2] = PR[90,2] + 42.761;
   1:L PR[91] R[100]mm/sec CNT100;
   1:  PR[91,1] = PR[90,1] + -1.119;
   1:  PR[91,2] = PR[90,2] + 41.867;
   1:L PR[91] R[100]mm/sec CNT100;
   1:  PR[91,1] = PR[90,1] + 6.250;
   1:L PR[91] R[100]mm/sec CNT100;
   1:  PR[91,1] = PR[90,1] + 5.356;
   1:  PR[91,2] = PR[90,2] + 42.761;
   1:L PR[91] R[100]mm/sec CNT100;
   1:  PR[91,1] = PR[90,1] + 3.853;
   1:  PR[91,2] = PR[90,2] + 48.367;
   1:L PR[91] R[100]mm/sec CNT100;
   1:  PR[91,1] = PR[90,1] + 5.356;
   1:  PR[91,2] = PR[90,2] + 53.973;
   1:L PR[91] R[100]mm/sec CNT100;
   1:  PR[91,1] = PR[90,1] + 6.250;
   1:  PR[91,2] = PR[90,2] + 54.867;
   1:L PR[91] R[100]mm/sec CNT100TB   .50sec,CALL END_PUD;
   1:  PR[92] = PR[91];
   1:  PR[92,3] = PR[92,3] + 50;
   1:J PR[92] 10% FINE;
   1:  PR[91,1] = PR[90,1] + 25.565;
   1:  PR[91,2] = PR[90,2] + 58.867;
   1:  PR[92] = PR[91];
   1:  PR[92,3] = PR[92,3] + 50;
   1:J PR[92] 10% FINE;
   1:L PR[91] R[100]mm/sec CNT100;
   1:  CALL LASER_DRAHT_START;
   1:  PR[91,1] = PR[90,1] + -20.435;
   1:L PR[91] R[100]mm/sec CNT100;
   1:  PR[91,2] = PR[90,2] + 37.867;
   1:L PR[91] R[100]mm/sec CNT100;
   1:  PR[91,1] = PR[90,1] + 25.565;
   1:L PR[91] R[100]mm/sec CNT100;
   1:  PR[91,2] = PR[90,2] + 58.867;
   1:L PR[91] R[100]mm/sec CNT100TB   .50sec,CALL END_PUD;
   1:  PR[92] = PR[91];
   1:  PR[92,3] = PR[92,3] + 50;
   1:J PR[92] 10% FINE;
   1:  PR[91,1] = PR[90,1] + 21.188;
   1:  PR[91,2] = PR[90,2] + 51.903;
   1:  PR[92] = PR[91];
   1:  PR[92,3] = PR[92,3] + 50;
   1:J PR[92] 10% FINE;
   1:L PR[91] R[100]mm/sec CNT100;
   1:  CALL LASER_DRAHT_START;
   1:  PR[91,1] = PR[90,1] + 22.136;
   1:  PR[91,2] = PR[90,2] + 48.367;
   1:L PR[91] R[100]mm/sec CNT100;
   1:  PR[91,1] = PR[90,1] + 21.188;
   1:  PR[91,2] = PR[90,2] + 44.832;
   1:L PR[91] R[100]mm/sec CNT100;
   1:  PR[91,1] = PR[90,1] + 18.601;
   1:  PR[91,2] = PR[90,2] + 42.244;
   1:L PR[91] R[100]mm/sec CNT100;
   1:  PR[91,1] = PR[90,1] + 15.065;
   1:  PR[91,2] = PR[90,2] + 41.296;
   1:L PR[91] R[100]mm/sec CNT100;
   1:  PR[91,1] = PR[90,1] + 11.530;
   1:  PR[91,2] = PR[90,2] + 42.244;
   1:L PR[91] R[100]mm/sec CNT100;
   1:  PR[91,1] = PR[90,1] + 8.942;
   1:  PR[91,2] = PR[90,2] + 44.832;
   1:L PR[91] R[100]mm/sec CNT100;
   1:  PR[91,1] = PR[90,1] + 7.995;
   1:  PR[91,2] = PR[90,2] + 48.367;
   1:L PR[91] R[100]mm/sec CNT100;
   1:  PR[91,1] = PR[90,1] + 8.942;
   1:  PR[91,2] = PR[90,2] + 51.903;
   1:L PR[91] R[100]mm/sec CNT100;
   1:  PR[91,1] = PR[90,1] + 11.530;
   1:  PR[91,2] = PR[90,2] + 54.490;
   1:L PR[91] R[100]mm/sec CNT100;
   1:  PR[91,1] = PR[90,1] + 15.065;
   1:  PR[91,2] = PR[90,2] + 55.438;
   1:L PR[91] R[100]mm/sec CNT100;
   1:  PR[91,1] = PR[90,1] + 18.601;
   1:  PR[91,2] = PR[90,2] + 54.490;
   1:L PR[91] R[100]mm/sec CNT100;
   1:  PR[91,1] = PR[90,1] + 21.188;
   1:  PR[91,2] = PR[90,2] + 51.903;
   1:L PR[91] R[100]mm/sec CNT100TB   .50sec,CALL END_PUD;
   1:  PR[92] = PR[91];
   1:  PR[92,3] = PR[92,3] + 50;
   1:J PR[92] 10% FINE;
   1:  PR[91,1] = PR[90,1] + -3.812;
   1:  PR[92] = PR[91];
   1:  PR[92,3] = PR[92,3] + 50;
   1:J PR[92] 10% FINE;
   1:L PR[91] R[100]mm/sec CNT100;
   1:  CALL LASER_DRAHT_START;
   1:  PR[91,1] = PR[90,1] + -2.864;
   1:  PR[91,2] = PR[90,2] + 48.367;
   1:L PR[91] R[100]mm/sec CNT100;
   1:  PR[91,1] = PR[90,1] + -3.812;
   1:  PR[91,2] = PR[90,2] + 44.832;
   1:L PR[91] R[100]mm/sec CNT100;
   1:  PR[91,1] = PR[90,1] + -6.399;
   1:  PR[91,2] = PR[90,2] + 42.244;
   1:L PR[91] R[100]mm/sec CNT100;
   1:  PR[91,1] = PR[90,1] + -9.935;
   1:  PR[91,2] = PR[90,2] + 41.296;
   1:L PR[91] R[100]mm/sec CNT100;
   1:  PR[91,1] = PR[90,1] + -13.470;
   1:  PR[91,2] = PR[90,2] + 42.244;
   1:L PR[91] R[100]mm/sec CNT100;
   1:  PR[91,1] = PR[90,1] + -16.058;
   1:  PR[91,2] = PR[90,2] + 44.832;
   1:L PR[91] R[100]mm/sec CNT100;
   1:  PR[91,1] = PR[90,1] + -17.005;
   1:  PR[91,2] = PR[90,2] + 48.367;
   1:L PR[91] R[100]mm/sec CNT100;
   1:  PR[91,1] = PR[90,1] + -16.058;
   1:  PR[91,2] = PR[90,2] + 51.903;
   1:L PR[91] R[100]mm/sec CNT100;
   1:  PR[91,1] = PR[90,1] + -13.470;
   1:  PR[91,2] = PR[90,2] + 54.490;
   1:L PR[91] R[100]mm/sec CNT100;
   1:  PR[91,1] = PR[90,1] + -9.935;
   1:  PR[91,2] = PR[90,2] + 55.438;
   1:L PR[91] R[100]mm/sec CNT100;
   1:  PR[91,1] = PR[90,1] + -6.399;
   1:  PR[91,2] = PR[90,2] + 54.490;
   1:L PR[91] R[100]mm/sec CNT100;
   1:  PR[91,1] = PR[90,1] + -3.812;
   1:  PR[91,2] = PR[90,2] + 51.903;
   1:L PR[91] R[100]mm/sec CNT100TB   .50sec,CALL END_PUD;
   1:  PR[92] = PR[91];
   1:  PR[92,3] = PR[92,3] + 50;
   1:J PR[92] 10% FINE;
   1:  PR[91] = PR[90];
   1:  PR[91,1] = PR[90,1] + 6.250;
   1:  PR[91,2] = PR[90,2] + 41.867;
   1:  PR[91,3] = PR[90,3] + 19.695;
   1:  PR[92] = PR[91];
   1:  PR[92,3] = PR[92,3] + 50;
   1:J PR[92] 10% FINE;
   1:L PR[91] R[100]mm/sec CNT100;
   1:  CALL LASER_DRAHT_START;
   1:  PR[91,1] = PR[90,1] + 5.356;
   1:  PR[91,2] = PR[90,2] + 42.761;
   1:L PR[91] R[100]mm/sec CNT100;
   1:  PR[91,1] = PR[90,1] + 3.854;
   1:  PR[91,2] = PR[90,2] + 48.367;
   1:L PR[91] R[100]mm/sec CNT100;
   1:  PR[91,1] = PR[90,1] + 5.356;
   1:  PR[91,2] = PR[90,2] + 53.973;
   1:L PR[91] R[100]mm/sec CNT100;
   1:  PR[91,1] = PR[90,1] + 6.250;
   1:  PR[91,2] = PR[90,2] + 54.867;
   1:L PR[91] R[100]mm/sec CNT100;
   1:  PR[91,1] = PR[90,1] + -1.119;
   1:L PR[91] R[100]mm/sec CNT100;
   1:  PR[91,1] = PR[90,1] + -0.225;
   1:  PR[91,2] = PR[90,2] + 53.973;
   1:L PR[91] R[100]mm/sec CNT100;
   1:  PR[91,1] = PR[90,1] + 1.277;
   1:  PR[91,2] = PR[90,2] + 48.367;
   1:L PR[91] R[100]mm/sec CNT100;
   1:  PR[91,1] = PR[90,1] + -0.225;
   1:  PR[91,2] = PR[90,2] + 42.761;
   1:L PR[91] R[100]mm/sec CNT100;
   1:  PR[91,1] = PR[90,1] + -1.119;
   1:  PR[91,2] = PR[90,2] + 41.867;
   1:L PR[91] R[100]mm/sec CNT100;
   1:  PR[91,1] = PR[90,1] + 6.250;
   1:L PR[91] R[100]mm/sec CNT100TB   .50sec,CALL END_PUD;
   1:  PR[92] = PR[91];
   1:  PR[92,3] = PR[92,3] + 50;
   1:J PR[92] 10% FINE;
   1:  PR[91,1] = PR[90,1] + 25.565;
   1:  PR[91,2] = PR[90,2] + 37.867;
   1:  PR[92] = PR[91];
   1:  PR[92,3] = PR[92,3] + 50;
   1:J PR[92] 10% FINE;
   1:L PR[91] R[100]mm/sec CNT100;
   1:  CALL LASER_DRAHT_START;
   1:  PR[91,2] = PR[90,2] + 58.867;
   1:L PR[91] R[100]mm/sec CNT100;
   1:  PR[91,1] = PR[90,1] + -20.435;
   1:L PR[91] R[100]mm/sec CNT100;
   1:  PR[91,2] = PR[90,2] + 37.867;
   1:L PR[91] R[100]mm/sec CNT100;
   1:  PR[91,1] = PR[90,1] + 25.565;
   1:L PR[91] R[100]mm/sec CNT100TB   .50sec,CALL END_PUD;
   1:  PR[92] = PR[91];
   1:  PR[92,3] = PR[92,3] + 50;
   1:J PR[92] 10% FINE;
   1:  PR[91,1] = PR[90,1] + 21.188;
   1:  PR[91,2] = PR[90,2] + 44.832;
   1:  PR[92] = PR[91];
   1:  PR[92,3] = PR[92,3] + 50;
   1:J PR[92] 10% FINE;
   1:L PR[91] R[100]mm/sec CNT100;
   1:  CALL LASER_DRAHT_START;
   1:  PR[91,1] = PR[90,1] + 18.601;
   1:  PR[91,2] = PR[90,2] + 42.244;
   1:L PR[91] R[100]mm/sec CNT100;
   1:  PR[91,1] = PR[90,1] + 15.065;
   1:  PR[91,2] = PR[90,2] + 41.296;
   1:L PR[91] R[100]mm/sec CNT100;
   1:  PR[91,1] = PR[90,1] + 11.530;
   1:  PR[91,2] = PR[90,2] + 42.244;
   1:L PR[91] R[100]mm/sec CNT100;
   1:  PR[91,1] = PR[90,1] + 8.942;
   1:  PR[91,2] = PR[90,2] + 44.832;
   1:L PR[91] R[100]mm/sec CNT100;
   1:  PR[91,1] = PR[90,1] + 7.995;
   1:  PR[91,2] = PR[90,2] + 48.367;
   1:L PR[91] R[100]mm/sec CNT100;
   1:  PR[91,1] = PR[90,1] + 8.942;
   1:  PR[91,2] = PR[90,2] + 51.903;
   1:L PR[91] R[100]mm/sec CNT100;
   1:  PR[91,1] = PR[90,1] + 11.530;
   1:  PR[91,2] = PR[90,2] + 54.490;
   1:L PR[91] R[100]mm/sec CNT100;
   1:  PR[91,1] = PR[90,1] + 15.065;
   1:  PR[91,2] = PR[90,2] + 55.438;
   1:L PR[91] R[100]mm/sec CNT100;
   1:  PR[91,1] = PR[90,1] + 18.601;
   1:  PR[91,2] = PR[90,2] + 54.490;
   1:L PR[91] R[100]mm/sec CNT100;
   1:  PR[91,1] = PR[90,1] + 21.188;
   1:  PR[91,2] = PR[90,2] + 51.903;
   1:L PR[91] R[100]mm/sec CNT100;
   1:  PR[91,1] = PR[90,1] + 22.136;
   1:  PR[91,2] = PR[90,2] + 48.367;
   1:L PR[91] R[100]mm/sec CNT100;
   1:  PR[91,1] = PR[90,1] + 21.188;
   1:  PR[91,2] = PR[90,2] + 44.832;
   1:L PR[91] R[100]mm/sec CNT100TB   .50sec,CALL END_PUD;
   1:  PR[92] = PR[91];
   1:  PR[92,3] = PR[92,3] + 50;
   1:J PR[92] 10% FINE;
   1:  PR[91,1] = PR[90,1] + -3.812;
   1:  PR[92] = PR[91];
   1:  PR[92,3] = PR[92,3] + 50;
   1:J PR[92] 10% FINE;
   1:L PR[91] R[100]mm/sec CNT100;
   1:  CALL LASER_DRAHT_START;
   1:  PR[91,1] = PR[90,1] + -6.399;
   1:  PR[91,2] = PR[90,2] + 42.244;
   1:L PR[91] R[100]mm/sec CNT100;
   1:  PR[91,1] = PR[90,1] + -9.935;
   1:  PR[91,2] = PR[90,2] + 41.296;
   1:L PR[91] R[100]mm/sec CNT100;
   1:  PR[91,1] = PR[90,1] + -13.470;
   1:  PR[91,2] = PR[90,2] + 42.244;
   1:L PR[91] R[100]mm/sec CNT100;
   1:  PR[91,1] = PR[90,1] + -16.058;
   1:  PR[91,2] = PR[90,2] + 44.832;
   1:L PR[91] R[100]mm/sec CNT100;
   1:  PR[91,1] = PR[90,1] + -17.005;
   1:  PR[91,2] = PR[90,2] + 48.367;
   1:L PR[91] R[100]mm/sec CNT100;
   1:  PR[91,1] = PR[90,1] + -16.058;
   1:  PR[91,2] = PR[90,2] + 51.903;
   1:L PR[91] R[100]mm/sec CNT100;
   1:  PR[91,1] = PR[90,1] + -13.470;
   1:  PR[91,2] = PR[90,2] + 54.490;
   1:L PR[91] R[100]mm/sec CNT100;
   1:  PR[91,1] = PR[90,1] + -9.935;
   1:  PR[91,2] = PR[90,2] + 55.438;
   1:L PR[91] R[100]mm/sec CNT100;
   1:  PR[91,1] = PR[90,1] + -6.399;
   1:  PR[91,2] = PR[90,2] + 54.490;
   1:L PR[91] R[100]mm/sec CNT100;
   1:  PR[91,1] = PR[90,1] + -3.812;
   1:  PR[91,2] = PR[90,2] + 51.903;
   1:L PR[91] R[100]mm/sec CNT100;
   1:  PR[91,1] = PR[90,1] + -2.864;
   1:  PR[91,2] = PR[90,2] + 48.367;
   1:L PR[91] R[100]mm/sec CNT100;
   1:  PR[91,1] = PR[90,1] + -3.812;
   1:  PR[91,2] = PR[90,2] + 44.832;
   1:L PR[91] R[100]mm/sec CNT100TB   .50sec,CALL END_PUD;
   1:  PR[92] = PR[91];
   1:  PR[92,3] = PR[92,3] + 50;
   1:J PR[92] 10% FINE;
   1:  PR[91] = PR[90];
   1:  PR[91,1] = PR[90,1] + -1.119;
   1:  PR[91,2] = PR[90,2] + 41.867;
   1:  PR[91,3] = PR[90,3] + 20.995;
   1:  PR[92] = PR[91];
   1:  PR[92,3] = PR[92,3] + 50;
   1:J PR[92] 10% FINE;
   1:L PR[91] R[100]mm/sec CNT100;
   1:  CALL LASER_DRAHT_START;
   1:  PR[91,1] = PR[90,1] + 6.250;
   1:L PR[91] R[100]mm/sec CNT100;
   1:  PR[91,1] = PR[90,1] + 5.356;
   1:  PR[91,2] = PR[90,2] + 42.761;
   1:L PR[91] R[100]mm/sec CNT100;
   1:  PR[91,1] = PR[90,1] + 3.854;
   1:  PR[91,2] = PR[90,2] + 48.367;
   1:L PR[91] R[100]mm/sec CNT100;
   1:  PR[91,1] = PR[90,1] + 5.356;
   1:  PR[91,2] = PR[90,2] + 53.973;
   1:L PR[91] R[100]mm/sec CNT100;
   1:  PR[91,1] = PR[90,1] + 6.250;
   1:  PR[91,2] = PR[90,2] + 54.867;
   1:L PR[91] R[100]mm/sec CNT100;
   1:  PR[91,1] = PR[90,1] + -1.119;
   1:L PR[91] R[100]mm/sec CNT100;
   1:  PR[91,1] = PR[90,1] + -0.225;
   1:  PR[91,2] = PR[90,2] + 53.973;
   1:L PR[91] R[100]mm/sec CNT100;
   1:  PR[91,1] = PR[90,1] + 1.277;
   1:  PR[91,2] = PR[90,2] + 48.367;
   1:L PR[91] R[100]mm/sec CNT100;
   1:  PR[91,1] = PR[90,1] + -0.225;
   1:  PR[91,2] = PR[90,2] + 42.761;
   1:L PR[91] R[100]mm/sec CNT100;
   1:  PR[91,1] = PR[90,1] + -1.119;
   1:  PR[91,2] = PR[90,2] + 41.867;
   1:L PR[91] R[100]mm/sec CNT100TB   .50sec,CALL END_PUD;
   1:  PR[92] = PR[91];
   1:  PR[92,3] = PR[92,3] + 50;
   1:J PR[92] 10% FINE;
   1:  PR[91,1] = PR[90,1] + -20.435;
   1:  PR[91,2] = PR[90,2] + 37.867;
   1:  PR[92] = PR[91];
   1:  PR[92,3] = PR[92,3] + 50;
   1:J PR[92] 10% FINE;
   1:L PR[91] R[100]mm/sec CNT100;
   1:  CALL LASER_DRAHT_START;
   1:  PR[91,1] = PR[90,1] + 25.565;
   1:L PR[91] R[100]mm/sec CNT100;
   1:  PR[91,2] = PR[90,2] + 58.867;
   1:L PR[91] R[100]mm/sec CNT100;
   1:  PR[91,1] = PR[90,1] + -20.435;
   1:L PR[91] R[100]mm/sec CNT100;
   1:  PR[91,2] = PR[90,2] + 37.867;
   1:L PR[91] R[100]mm/sec CNT100TB   .50sec,CALL END_PUD;
   1:  PR[92] = PR[91];
   1:  PR[92,3] = PR[92,3] + 50;
   1:J PR[92] 10% FINE;
   1:  PR[91,1] = PR[90,1] + -16.058;
   1:  PR[91,2] = PR[90,2] + 44.832;
   1:  PR[92] = PR[91];
   1:  PR[92,3] = PR[92,3] + 50;
   1:J PR[92] 10% FINE;
   1:L PR[91] R[100]mm/sec CNT100;
   1:  CALL LASER_DRAHT_START;
   1:  PR[91,1] = PR[90,1] + -17.005;
   1:  PR[91,2] = PR[90,2] + 48.367;
   1:L PR[91] R[100]mm/sec CNT100;
   1:  PR[91,1] = PR[90,1] + -16.058;
   1:  PR[91,2] = PR[90,2] + 51.902;
   1:L PR[91] R[100]mm/sec CNT100;
   1:  PR[91,1] = PR[90,1] + -13.470;
   1:  PR[91,2] = PR[90,2] + 54.490;
   1:L PR[91] R[100]mm/sec CNT100;
   1:  PR[91,1] = PR[90,1] + -9.935;
   1:  PR[91,2] = PR[90,2] + 55.438;
   1:L PR[91] R[100]mm/sec CNT100;
   1:  PR[91,1] = PR[90,1] + -6.399;
   1:  PR[91,2] = PR[90,2] + 54.490;
   1:L PR[91] R[100]mm/sec CNT100;
   1:  PR[91,1] = PR[90,1] + -3.812;
   1:  PR[91,2] = PR[90,2] + 51.902;
   1:L PR[91] R[100]mm/sec CNT100;
   1:  PR[91,1] = PR[90,1] + -2.864;
   1:  PR[91,2] = PR[90,2] + 48.367;
   1:L PR[91] R[100]mm/sec CNT100;
   1:  PR[91,1] = PR[90,1] + -3.812;
   1:  PR[91,2] = PR[90,2] + 44.832;
   1:L PR[91] R[100]mm/sec CNT100;
   1:  PR[91,1] = PR[90,1] + -6.399;
   1:  PR[91,2] = PR[90,2] + 42.244;
   1:L PR[91] R[100]mm/sec CNT100;
   1:  PR[91,1] = PR[90,1] + -9.935;
   1:  PR[91,2] = PR[90,2] + 41.296;
   1:L PR[91] R[100]mm/sec CNT100;
   1:  PR[91,1] = PR[90,1] + -13.470;
   1:  PR[91,2] = PR[90,2] + 42.244;
   1:L PR[91] R[100]mm/sec CNT100;
   1:  PR[91,1] = PR[90,1] + -16.058;
   1:  PR[91,2] = PR[90,2] + 44.832;
   1:L PR[91] R[100]mm/sec CNT100TB   .50sec,CALL END_PUD;
   1:  PR[92] = PR[91];
   1:  PR[92,3] = PR[92,3] + 50;
   1:J PR[92] 10% FINE;
   1:  PR[91,1] = PR[90,1] + 8.942;
   1:  PR[92] = PR[91];
   1:  PR[92,3] = PR[92,3] + 50;
   1:J PR[92] 10% FINE;
   1:L PR[91] R[100]mm/sec CNT100;
   1:  CALL LASER_DRAHT_START;
   1:  PR[91,1] = PR[90,1] + 7.995;
   1:  PR[91,2] = PR[90,2] + 48.367;
   1:L PR[91] R[100]mm/sec CNT100;
   1:  PR[91,1] = PR[90,1] + 8.942;
   1:  PR[91,2] = PR[90,2] + 51.902;
   1:L PR[91] R[100]mm/sec CNT100;
   1:  PR[91,1] = PR[90,1] + 11.530;
   1:  PR[91,2] = PR[90,2] + 54.490;
   1:L PR[91] R[100]mm/sec CNT100;
   1:  PR[91,1] = PR[90,1] + 15.065;
   1:  PR[91,2] = PR[90,2] + 55.438;
   1:L PR[91] R[100]mm/sec CNT100;
   1:  PR[91,1] = PR[90,1] + 18.601;
   1:  PR[91,2] = PR[90,2] + 54.490;
   1:L PR[91] R[100]mm/sec CNT100;
   1:  PR[91,1] = PR[90,1] + 21.188;
   1:  PR[91,2] = PR[90,2] + 51.902;
   1:L PR[91] R[100]mm/sec CNT100;
   1:  PR[91,1] = PR[90,1] + 22.136;
   1:  PR[91,2] = PR[90,2] + 48.367;
   1:L PR[91] R[100]mm/sec CNT100;
   1:  PR[91,1] = PR[90,1] + 21.188;
   1:  PR[91,2] = PR[90,2] + 44.832;
   1:L PR[91] R[100]mm/sec CNT100;
   1:  PR[91,1] = PR[90,1] + 18.601;
   1:  PR[91,2] = PR[90,2] + 42.244;
   1:L PR[91] R[100]mm/sec CNT100;
   1:  PR[91,1] = PR[90,1] + 15.065;
   1:  PR[91,2] = PR[90,2] + 41.296;
   1:L PR[91] R[100]mm/sec CNT100;
   1:  PR[91,1] = PR[90,1] + 11.530;
   1:  PR[91,2] = PR[90,2] + 42.244;
   1:L PR[91] R[100]mm/sec CNT100;
   1:  PR[91,1] = PR[90,1] + 8.942;
   1:  PR[91,2] = PR[90,2] + 44.832;
   1:L PR[91] R[100]mm/sec CNT100TB   .50sec,CALL END_PUD;
   1:  PR[92] = PR[91];
   1:  PR[92,3] = PR[92,3] + 50;
   1:J PR[92] 10% FINE;
   1:  PR[91] = PR[90];
   1:  PR[91,1] = PR[90,1] + -1.119;
   1:  PR[91,2] = PR[90,2] + 41.867;
   1:  PR[91,3] = PR[90,3] + 22.295;
   1:  PR[92] = PR[91];
   1:  PR[92,3] = PR[92,3] + 50;
   1:J PR[92] 10% FINE;
   1:L PR[91] R[100]mm/sec CNT100;
   1:  CALL LASER_DRAHT_START;
   1:  PR[91,1] = PR[90,1] + 6.250;
   1:L PR[91] R[100]mm/sec CNT100;
   1:  PR[91,1] = PR[90,1] + 5.356;
   1:  PR[91,2] = PR[90,2] + 42.761;
   1:L PR[91] R[100]mm/sec CNT100;
   1:  PR[91,1] = PR[90,1] + 3.854;
   1:  PR[91,2] = PR[90,2] + 48.367;
   1:L PR[91] R[100]mm/sec CNT100;
   1:  PR[91,1] = PR[90,1] + 5.356;
   1:  PR[91,2] = PR[90,2] + 53.973;
   1:L PR[91] R[100]mm/sec CNT100;
   1:  PR[91,1] = PR[90,1] + 6.250;
   1:  PR[91,2] = PR[90,2] + 54.867;
   1:L PR[91] R[100]mm/sec CNT100;
   1:  PR[91,1] = PR[90,1] + -1.119;
   1:L PR[91] R[100]mm/sec CNT100;
   1:  PR[91,1] = PR[90,1] + -0.225;
   1:  PR[91,2] = PR[90,2] + 53.973;
   1:L PR[91] R[100]mm/sec CNT100;
   1:  PR[91,1] = PR[90,1] + 1.277;
   1:  PR[91,2] = PR[90,2] + 48.367;
   1:L PR[91] R[100]mm/sec CNT100;
   1:  PR[91,1] = PR[90,1] + -0.225;
   1:  PR[91,2] = PR[90,2] + 42.761;
   1:L PR[91] R[100]mm/sec CNT100;
   1:  PR[91,1] = PR[90,1] + -1.119;
   1:  PR[91,2] = PR[90,2] + 41.867;
   1:L PR[91] R[100]mm/sec CNT100TB   .50sec,CALL END_PUD;
   1:  PR[92] = PR[91];
   1:  PR[92,3] = PR[92,3] + 50;
   1:J PR[92] 10% FINE;
   1:  PR[91,1] = PR[90,1] + -20.435;
   1:  PR[91,2] = PR[90,2] + 37.867;
   1:  PR[92] = PR[91];
   1:  PR[92,3] = PR[92,3] + 50;
   1:J PR[92] 10% FINE;
   1:L PR[91] R[100]mm/sec CNT100;
   1:  CALL LASER_DRAHT_START;
   1:  PR[91,1] = PR[90,1] + 25.565;
   1:L PR[91] R[100]mm/sec CNT100;
   1:  PR[91,2] = PR[90,2] + 58.867;
   1:L PR[91] R[100]mm/sec CNT100;
   1:  PR[91,1] = PR[90,1] + -20.435;
   1:L PR[91] R[100]mm/sec CNT100;
   1:  PR[91,2] = PR[90,2] + 37.867;
   1:L PR[91] R[100]mm/sec CNT100TB   .50sec,CALL END_PUD;
   1:  PR[92] = PR[91];
   1:  PR[92,3] = PR[92,3] + 50;
   1:J PR[92] 10% FINE;
   1:  PR[91,1] = PR[90,1] + -16.058;
   1:  PR[91,2] = PR[90,2] + 44.832;
   1:  PR[92] = PR[91];
   1:  PR[92,3] = PR[92,3] + 50;
   1:J PR[92] 10% FINE;
   1:L PR[91] R[100]mm/sec CNT100;
   1:  CALL LASER_DRAHT_START;
   1:  PR[91,1] = PR[90,1] + -17.005;
   1:  PR[91,2] = PR[90,2] + 48.367;
   1:L PR[91] R[100]mm/sec CNT100;
   1:  PR[91,1] = PR[90,1] + -16.058;
   1:  PR[91,2] = PR[90,2] + 51.902;
   1:L PR[91] R[100]mm/sec CNT100;
   1:  PR[91,1] = PR[90,1] + -13.470;
   1:  PR[91,2] = PR[90,2] + 54.490;
   1:L PR[91] R[100]mm/sec CNT100;
   1:  PR[91,1] = PR[90,1] + -9.935;
   1:  PR[91,2] = PR[90,2] + 55.438;
   1:L PR[91] R[100]mm/sec CNT100;
   1:  PR[91,1] = PR[90,1] + -6.399;
   1:  PR[91,2] = PR[90,2] + 54.490;
   1:L PR[91] R[100]mm/sec CNT100;
   1:  PR[91,1] = PR[90,1] + -3.812;
   1:  PR[91,2] = PR[90,2] + 51.902;
   1:L PR[91] R[100]mm/sec CNT100;
   1:  PR[91,1] = PR[90,1] + -2.864;
   1:  PR[91,2] = PR[90,2] + 48.367;
   1:L PR[91] R[100]mm/sec CNT100;
   1:  PR[91,1] = PR[90,1] + -3.812;
   1:  PR[91,2] = PR[90,2] + 44.832;
   1:L PR[91] R[100]mm/sec CNT100;
   1:  PR[91,1] = PR[90,1] + -6.399;
   1:  PR[91,2] = PR[90,2] + 42.244;
   1:L PR[91] R[100]mm/sec CNT100;
   1:  PR[91,1] = PR[90,1] + -9.935;
   1:  PR[91,2] = PR[90,2] + 41.296;
   1:L PR[91] R[100]mm/sec CNT100;
   1:  PR[91,1] = PR[90,1] + -13.470;
   1:  PR[91,2] = PR[90,2] + 42.244;
   1:L PR[91] R[100]mm/sec CNT100;
   1:  PR[91,1] = PR[90,1] + -16.058;
   1:  PR[91,2] = PR[90,2] + 44.832;
   1:L PR[91] R[100]mm/sec CNT100TB   .50sec,CALL END_PUD;
   1:  PR[92] = PR[91];
   1:  PR[92,3] = PR[92,3] + 50;
   1:J PR[92] 10% FINE;
   1:  PR[91,1] = PR[90,1] + 8.942;
   1:  PR[92] = PR[91];
   1:  PR[92,3] = PR[92,3] + 50;
   1:J PR[92] 10% FINE;
   1:L PR[91] R[100]mm/sec CNT100;
   1:  CALL LASER_DRAHT_START;
   1:  PR[91,1] = PR[90,1] + 7.995;
   1:  PR[91,2] = PR[90,2] + 48.367;
   1:L PR[91] R[100]mm/sec CNT100;
   1:  PR[91,1] = PR[90,1] + 8.942;
   1:  PR[91,2] = PR[90,2] + 51.902;
   1:L PR[91] R[100]mm/sec CNT100;
   1:  PR[91,1] = PR[90,1] + 11.530;
   1:  PR[91,2] = PR[90,2] + 54.490;
   1:L PR[91] R[100]mm/sec CNT100;
   1:  PR[91,1] = PR[90,1] + 15.065;
   1:  PR[91,2] = PR[90,2] + 55.438;
   1:L PR[91] R[100]mm/sec CNT100;
   1:  PR[91,1] = PR[90,1] + 18.601;
   1:  PR[91,2] = PR[90,2] + 54.490;
   1:L PR[91] R[100]mm/sec CNT100;
   1:  PR[91,1] = PR[90,1] + 21.188;
   1:  PR[91,2] = PR[90,2] + 51.902;
   1:L PR[91] R[100]mm/sec CNT100;
   1:  PR[91,1] = PR[90,1] + 22.136;
   1:  PR[91,2] = PR[90,2] + 48.367;
   1:L PR[91] R[100]mm/sec CNT100;
   1:  PR[91,1] = PR[90,1] + 21.188;
   1:  PR[91,2] = PR[90,2] + 44.832;
   1:L PR[91] R[100]mm/sec CNT100;
   1:  PR[91,1] = PR[90,1] + 18.601;
   1:  PR[91,2] = PR[90,2] + 42.244;
   1:L PR[91] R[100]mm/sec CNT100;
   1:  PR[91,1] = PR[90,1] + 15.065;
   1:  PR[91,2] = PR[90,2] + 41.296;
   1:L PR[91] R[100]mm/sec CNT100;
   1:  PR[91,1] = PR[90,1] + 11.530;
   1:  PR[91,2] = PR[90,2] + 42.244;
   1:L PR[91] R[100]mm/sec CNT100;
   1:  PR[91,1] = PR[90,1] + 8.942;
   1:  PR[91,2] = PR[90,2] + 44.832;
   1:L PR[91] R[100]mm/sec CNT100TB   .50sec,CALL END_PUD;
   1:  PR[92] = PR[91];
   1:  PR[92,3] = PR[92,3] + 50;
   1:J PR[92] 10% FINE;
   1:  PR[91] = PR[90];
   1:  PR[91,1] = PR[90,1] + 6.250;
   1:  PR[91,2] = PR[90,2] + 54.867;
   1:  PR[91,3] = PR[90,3] + 23.595;
   1:  PR[92] = PR[91];
   1:  PR[92,3] = PR[92,3] + 50;
   1:J PR[92] 10% FINE;
   1:L PR[91] R[100]mm/sec CNT100;
   1:  CALL LASER_DRAHT_START;
   1:  PR[91,1] = PR[90,1] + -1.119;
   1:L PR[91] R[100]mm/sec CNT100;
   1:  PR[91,1] = PR[90,1] + -0.225;
   1:  PR[91,2] = PR[90,2] + 53.973;
   1:L PR[91] R[100]mm/sec CNT100;
   1:  PR[91,1] = PR[90,1] + 1.277;
   1:  PR[91,2] = PR[90,2] + 48.367;
   1:L PR[91] R[100]mm/sec CNT100;
   1:  PR[91,1] = PR[90,1] + -0.225;
   1:  PR[91,2] = PR[90,2] + 42.761;
   1:L PR[91] R[100]mm/sec CNT100;
   1:  PR[91,1] = PR[90,1] + -1.119;
   1:  PR[91,2] = PR[90,2] + 41.867;
   1:L PR[91] R[100]mm/sec CNT100;
   1:  PR[91,1] = PR[90,1] + 6.250;
   1:L PR[91] R[100]mm/sec CNT100;
   1:  PR[91,1] = PR[90,1] + 5.356;
   1:  PR[91,2] = PR[90,2] + 42.761;
   1:L PR[91] R[100]mm/sec CNT100;
   1:  PR[91,1] = PR[90,1] + 3.854;
   1:  PR[91,2] = PR[90,2] + 48.367;
   1:L PR[91] R[100]mm/sec CNT100;
   1:  PR[91,1] = PR[90,1] + 5.356;
   1:  PR[91,2] = PR[90,2] + 53.973;
   1:L PR[91] R[100]mm/sec CNT100;
   1:  PR[91,1] = PR[90,1] + 6.250;
   1:  PR[91,2] = PR[90,2] + 54.867;
   1:L PR[91] R[100]mm/sec CNT100TB   .50sec,CALL END_PUD;
   1:  PR[92] = PR[91];
   1:  PR[92,3] = PR[92,3] + 50;
   1:J PR[92] 10% FINE;
   1:  PR[91,1] = PR[90,1] + 25.565;
   1:  PR[91,2] = PR[90,2] + 58.867;
   1:  PR[92] = PR[91];
   1:  PR[92,3] = PR[92,3] + 50;
   1:J PR[92] 10% FINE;
   1:L PR[91] R[100]mm/sec CNT100;
   1:  CALL LASER_DRAHT_START;
   1:  PR[91,1] = PR[90,1] + -20.435;
   1:L PR[91] R[100]mm/sec CNT100;
   1:  PR[91,2] = PR[90,2] + 37.867;
   1:L PR[91] R[100]mm/sec CNT100;
   1:  PR[91,1] = PR[90,1] + 25.565;
   1:L PR[91] R[100]mm/sec CNT100;
   1:  PR[91,2] = PR[90,2] + 58.867;
   1:L PR[91] R[100]mm/sec CNT100TB   .50sec,CALL END_PUD;
   1:  PR[92] = PR[91];
   1:  PR[92,3] = PR[92,3] + 50;
   1:J PR[92] 10% FINE;
   1:  PR[91,1] = PR[90,1] + 21.188;
   1:  PR[91,2] = PR[90,2] + 51.902;
   1:  PR[92] = PR[91];
   1:  PR[92,3] = PR[92,3] + 50;
   1:J PR[92] 10% FINE;
   1:L PR[91] R[100]mm/sec CNT100;
   1:  CALL LASER_DRAHT_START;
   1:  PR[91,1] = PR[90,1] + 22.136;
   1:  PR[91,2] = PR[90,2] + 48.367;
   1:L PR[91] R[100]mm/sec CNT100;
   1:  PR[91,1] = PR[90,1] + 21.188;
   1:  PR[91,2] = PR[90,2] + 44.832;
   1:L PR[91] R[100]mm/sec CNT100;
   1:  PR[91,1] = PR[90,1] + 18.601;
   1:  PR[91,2] = PR[90,2] + 42.244;
   1:L PR[91] R[100]mm/sec CNT100;
   1:  PR[91,1] = PR[90,1] + 15.065;
   1:  PR[91,2] = PR[90,2] + 41.296;
   1:L PR[91] R[100]mm/sec CNT100;
   1:  PR[91,1] = PR[90,1] + 11.530;
   1:  PR[91,2] = PR[90,2] + 42.244;
   1:L PR[91] R[100]mm/sec CNT100;
   1:  PR[91,1] = PR[90,1] + 8.942;
   1:  PR[91,2] = PR[90,2] + 44.832;
   1:L PR[91] R[100]mm/sec CNT100;
   1:  PR[91,1] = PR[90,1] + 7.995;
   1:  PR[91,2] = PR[90,2] + 48.367;
   1:L PR[91] R[100]mm/sec CNT100;
   1:  PR[91,1] = PR[90,1] + 8.942;
   1:  PR[91,2] = PR[90,2] + 51.902;
   1:L PR[91] R[100]mm/sec CNT100;
   1:  PR[91,1] = PR[90,1] + 11.530;
   1:  PR[91,2] = PR[90,2] + 54.490;
   1:L PR[91] R[100]mm/sec CNT100;
   1:  PR[91,1] = PR[90,1] + 15.065;
   1:  PR[91,2] = PR[90,2] + 55.438;
   1:L PR[91] R[100]mm/sec CNT100;
   1:  PR[91,1] = PR[90,1] + 18.601;
   1:  PR[91,2] = PR[90,2] + 54.490;
   1:L PR[91] R[100]mm/sec CNT100;
   1:  PR[91,1] = PR[90,1] + 21.188;
   1:  PR[91,2] = PR[90,2] + 51.902;
   1:L PR[91] R[100]mm/sec CNT100TB   .50sec,CALL END_PUD;
   1:  PR[92] = PR[91];
   1:  PR[92,3] = PR[92,3] + 50;
   1:J PR[92] 10% FINE;
   1:  PR[91,1] = PR[90,1] + -3.812;
   1:  PR[92] = PR[91];
   1:  PR[92,3] = PR[92,3] + 50;
   1:J PR[92] 10% FINE;
   1:L PR[91] R[100]mm/sec CNT100;
   1:  CALL LASER_DRAHT_START;
   1:  PR[91,1] = PR[90,1] + -2.864;
   1:  PR[91,2] = PR[90,2] + 48.367;
   1:L PR[91] R[100]mm/sec CNT100;
   1:  PR[91,1] = PR[90,1] + -3.812;
   1:  PR[91,2] = PR[90,2] + 44.832;
   1:L PR[91] R[100]mm/sec CNT100;
   1:  PR[91,1] = PR[90,1] + -6.399;
   1:  PR[91,2] = PR[90,2] + 42.244;
   1:L PR[91] R[100]mm/sec CNT100;
   1:  PR[91,1] = PR[90,1] + -9.935;
   1:  PR[91,2] = PR[90,2] + 41.296;
   1:L PR[91] R[100]mm/sec CNT100;
   1:  PR[91,1] = PR[90,1] + -13.470;
   1:  PR[91,2] = PR[90,2] + 42.244;
   1:L PR[91] R[100]mm/sec CNT100;
   1:  PR[91,1] = PR[90,1] + -16.058;
   1:  PR[91,2] = PR[90,2] + 44.832;
   1:L PR[91] R[100]mm/sec CNT100;
   1:  PR[91,1] = PR[90,1] + -17.005;
   1:  PR[91,2] = PR[90,2] + 48.367;
   1:L PR[91] R[100]mm/sec CNT100;
   1:  PR[91,1] = PR[90,1] + -16.058;
   1:  PR[91,2] = PR[90,2] + 51.902;
   1:L PR[91] R[100]mm/sec CNT100;
   1:  PR[91,1] = PR[90,1] + -13.470;
   1:  PR[91,2] = PR[90,2] + 54.490;
   1:L PR[91] R[100]mm/sec CNT100;
   1:  PR[91,1] = PR[90,1] + -9.935;
   1:  PR[91,2] = PR[90,2] + 55.438;
   1:L PR[91] R[100]mm/sec CNT100;
   1:  PR[91,1] = PR[90,1] + -6.399;
   1:  PR[91,2] = PR[90,2] + 54.490;
   1:L PR[91] R[100]mm/sec CNT100;
   1:  PR[91,1] = PR[90,1] + -3.812;
   1:  PR[91,2] = PR[90,2] + 51.902;
   1:L PR[91] R[100]mm/sec CNT100TB   .50sec,CALL END_PUD;
   1:  PR[92] = PR[91];
   1:  PR[92,3] = PR[92,3] + 50;
   1:J PR[92] 10% FINE;
   1:  PR[91] = PR[90];
   1:  PR[91,1] = PR[90,1] + 6.250;
   1:  PR[91,2] = PR[90,2] + 41.867;
   1:  PR[91,3] = PR[90,3] + 24.895;
   1:  PR[92] = PR[91];
   1:  PR[92,3] = PR[92,3] + 50;
   1:J PR[92] 10% FINE;
   1:L PR[91] R[100]mm/sec CNT100;
   1:  CALL LASER_DRAHT_START;
   1:  PR[91,1] = PR[90,1] + 5.356;
   1:  PR[91,2] = PR[90,2] + 42.761;
   1:L PR[91] R[100]mm/sec CNT100;
   1:  PR[91,1] = PR[90,1] + 3.854;
   1:  PR[91,2] = PR[90,2] + 48.367;
   1:L PR[91] R[100]mm/sec CNT100;
   1:  PR[91,1] = PR[90,1] + 5.356;
   1:  PR[91,2] = PR[90,2] + 53.973;
   1:L PR[91] R[100]mm/sec CNT100;
   1:  PR[91,1] = PR[90,1] + 6.250;
   1:  PR[91,2] = PR[90,2] + 54.867;
   1:L PR[91] R[100]mm/sec CNT100;
   1:  PR[91,1] = PR[90,1] + -1.119;
   1:L PR[91] R[100]mm/sec CNT100;
   1:  PR[91,1] = PR[90,1] + -0.225;
   1:  PR[91,2] = PR[90,2] + 53.973;
   1:L PR[91] R[100]mm/sec CNT100;
   1:  PR[91,1] = PR[90,1] + 1.277;
   1:  PR[91,2] = PR[90,2] + 48.367;
   1:L PR[91] R[100]mm/sec CNT100;
   1:  PR[91,1] = PR[90,1] + -0.225;
   1:  PR[91,2] = PR[90,2] + 42.761;
   1:L PR[91] R[100]mm/sec CNT100;
   1:  PR[91,1] = PR[90,1] + -1.119;
   1:  PR[91,2] = PR[90,2] + 41.867;
   1:L PR[91] R[100]mm/sec CNT100;
   1:  PR[91,1] = PR[90,1] + 6.250;
   1:L PR[91] R[100]mm/sec CNT100TB   .50sec,CALL END_PUD;
   1:  PR[92] = PR[91];
   1:  PR[92,3] = PR[92,3] + 50;
   1:J PR[92] 10% FINE;
   1:  PR[91,1] = PR[90,1] + 25.565;
   1:  PR[91,2] = PR[90,2] + 37.867;
   1:  PR[92] = PR[91];
   1:  PR[92,3] = PR[92,3] + 50;
   1:J PR[92] 10% FINE;
   1:L PR[91] R[100]mm/sec CNT100;
   1:  CALL LASER_DRAHT_START;
   1:  PR[91,2] = PR[90,2] + 58.867;
   1:L PR[91] R[100]mm/sec CNT100;
   1:  PR[91,1] = PR[90,1] + -20.435;
   1:L PR[91] R[100]mm/sec CNT100;
   1:  PR[91,2] = PR[90,2] + 37.867;
   1:L PR[91] R[100]mm/sec CNT100;
   1:  PR[91,1] = PR[90,1] + 25.565;
   1:L PR[91] R[100]mm/sec CNT100TB   .50sec,CALL END_PUD;
   1:  PR[92] = PR[91];
   1:  PR[92,3] = PR[92,3] + 50;
   1:J PR[92] 10% FINE;
   1:  PR[91,1] = PR[90,1] + 21.188;
   1:  PR[91,2] = PR[90,2] + 44.832;
   1:  PR[92] = PR[91];
   1:  PR[92,3] = PR[92,3] + 50;
   1:J PR[92] 10% FINE;
   1:L PR[91] R[100]mm/sec CNT100;
   1:  CALL LASER_DRAHT_START;
   1:  PR[91,1] = PR[90,1] + 18.601;
   1:  PR[91,2] = PR[90,2] + 42.244;
   1:L PR[91] R[100]mm/sec CNT100;
   1:  PR[91,1] = PR[90,1] + 15.065;
   1:  PR[91,2] = PR[90,2] + 41.297;
   1:L PR[91] R[100]mm/sec CNT100;
   1:  PR[91,1] = PR[90,1] + 11.530;
   1:  PR[91,2] = PR[90,2] + 42.244;
   1:L PR[91] R[100]mm/sec CNT100;
   1:  PR[91,1] = PR[90,1] + 8.942;
   1:  PR[91,2] = PR[90,2] + 44.832;
   1:L PR[91] R[100]mm/sec CNT100;
   1:  PR[91,1] = PR[90,1] + 7.995;
   1:  PR[91,2] = PR[90,2] + 48.367;
   1:L PR[91] R[100]mm/sec CNT100;
   1:  PR[91,1] = PR[90,1] + 8.942;
   1:  PR[91,2] = PR[90,2] + 51.902;
   1:L PR[91] R[100]mm/sec CNT100;
   1:  PR[91,1] = PR[90,1] + 11.530;
   1:  PR[91,2] = PR[90,2] + 54.490;
   1:L PR[91] R[100]mm/sec CNT100;
   1:  PR[91,1] = PR[90,1] + 15.065;
   1:  PR[91,2] = PR[90,2] + 55.438;
   1:L PR[91] R[100]mm/sec CNT100;
   1:  PR[91,1] = PR[90,1] + 18.601;
   1:  PR[91,2] = PR[90,2] + 54.490;
   1:L PR[91] R[100]mm/sec CNT100;
   1:  PR[91,1] = PR[90,1] + 21.188;
   1:  PR[91,2] = PR[90,2] + 51.902;
   1:L PR[91] R[100]mm/sec CNT100;
   1:  PR[91,1] = PR[90,1] + 22.136;
   1:  PR[91,2] = PR[90,2] + 48.367;
   1:L PR[91] R[100]mm/sec CNT100;
   1:  PR[91,1] = PR[90,1] + 21.188;
   1:  PR[91,2] = PR[90,2] + 44.832;
   1:L PR[91] R[100]mm/sec CNT100TB   .50sec,CALL END_PUD;
   1:  PR[92] = PR[91];
   1:  PR[92,3] = PR[92,3] + 50;
   1:J PR[92] 10% FINE;
   1:  PR[91,1] = PR[90,1] + -3.812;
   1:  PR[92] = PR[91];
   1:  PR[92,3] = PR[92,3] + 50;
   1:J PR[92] 10% FINE;
   1:L PR[91] R[100]mm/sec CNT100;
   1:  CALL LASER_DRAHT_START;
   1:  PR[91,1] = PR[90,1] + -6.399;
   1:  PR[91,2] = PR[90,2] + 42.244;
   1:L PR[91] R[100]mm/sec CNT100;
   1:  PR[91,1] = PR[90,1] + -9.935;
   1:  PR[91,2] = PR[90,2] + 41.297;
   1:L PR[91] R[100]mm/sec CNT100;
   1:  PR[91,1] = PR[90,1] + -13.470;
   1:  PR[91,2] = PR[90,2] + 42.244;
   1:L PR[91] R[100]mm/sec CNT100;
   1:  PR[91,1] = PR[90,1] + -16.058;
   1:  PR[91,2] = PR[90,2] + 44.832;
   1:L PR[91] R[100]mm/sec CNT100;
   1:  PR[91,1] = PR[90,1] + -17.005;
   1:  PR[91,2] = PR[90,2] + 48.367;
   1:L PR[91] R[100]mm/sec CNT100;
   1:  PR[91,1] = PR[90,1] + -16.058;
   1:  PR[91,2] = PR[90,2] + 51.902;
   1:L PR[91] R[100]mm/sec CNT100;
   1:  PR[91,1] = PR[90,1] + -13.470;
   1:  PR[91,2] = PR[90,2] + 54.490;
   1:L PR[91] R[100]mm/sec CNT100;
   1:  PR[91,1] = PR[90,1] + -9.935;
   1:  PR[91,2] = PR[90,2] + 55.438;
   1:L PR[91] R[100]mm/sec CNT100;
   1:  PR[91,1] = PR[90,1] + -6.399;
   1:  PR[91,2] = PR[90,2] + 54.490;
   1:L PR[91] R[100]mm/sec CNT100;
   1:  PR[91,1] = PR[90,1] + -3.812;
   1:  PR[91,2] = PR[90,2] + 51.902;
   1:L PR[91] R[100]mm/sec CNT100;
   1:  PR[91,1] = PR[90,1] + -2.864;
   1:  PR[91,2] = PR[90,2] + 48.367;
   1:L PR[91] R[100]mm/sec CNT100;
   1:  PR[91,1] = PR[90,1] + -3.812;
